DATA_BLOCK "ShiftmodelInterfaceHmi"   // DB103
TITLE = Schichtzeiten / ShiftmodelTimes
AUTHOR : SICAR
FAMILY : Shiftmodel
VERSION : 1.0
// Global DB fuer Schnittstelle HMI / Global DB for HMI interface
// stored: InstanceOfName LSicar_typeShiftmodelHmi, InstanceOfType UDT
"LSicar_typeShiftmodelHmi"
   // VAR RETAIN
   //    shiftTimesListIndex : DInt := 1;
   //    actualTimesDay : Array[0..7] of "LSicar_typeShiftmodTime1Day";
   //    actualSignalsDay : Array[0..7] of "LSicar_typeShiftmodSign1Day";
   //    summary : "LSicar_typeShiftmodSumHmi";
   //    actualDay : USInt := 0;
   //    shiftTimesListOnOff : Bool := TRUE;   // Schichtzeiten Remote OnOff / Shift times OnOff
   //    setAdjTimes : Bool := FALSE;
   //    hmiTimesValidFor : Array[0..3] of "LSicar_typeWeekdayBools";
   //    hmiTimes : Array[0..3] of "LSicar_typeShiftmodTime1Shift";   // Schnittstelle Lokale Zeiten (eingeben am HMI) / Interface Local Times (Input on HMI)
   //    productionTimes : "LSicar_typeProdTimesHmi";
   // END_VAR
BEGIN
   actualTimesDay[0].shift[0..3].endCircuitTime := TOD#00:00:00;
   actualTimesDay[1].shift[0..3].endCircuitTime := TOD#00:00:00;
   actualTimesDay[2].shift[0..3].endCircuitTime := TOD#00:00:00;
   actualTimesDay[3].shift[0..3].endCircuitTime := TOD#00:00:00;
   actualTimesDay[4].shift[0..3].endCircuitTime := TOD#00:00:00;
   actualTimesDay[5].shift[0..3].endCircuitTime := TOD#00:00:00;
   actualTimesDay[6].shift[0..3].endCircuitTime := TOD#00:00:00;
   actualTimesDay[7].shift[0..3].endCircuitTime := TOD#00:00:00;
   actualTimesDay[0].shift[0..3].start := TOD#00:00:00;
   actualTimesDay[1].shift[0..3].start := TOD#00:00:00;
   actualTimesDay[2].shift[0..3].start := TOD#00:00:00;
   actualTimesDay[3].shift[0..3].start := TOD#00:00:00;
   actualTimesDay[4].shift[0..3].start := TOD#00:00:00;
   actualTimesDay[5].shift[0..3].start := TOD#00:00:00;
   actualTimesDay[6].shift[0..3].start := TOD#00:00:00;
   actualTimesDay[7].shift[0..3].start := TOD#00:00:00;
   actualTimesDay[0].shift[0].break[0..4].start := TOD#00:00:00;
   actualTimesDay[0].shift[1].break[0..4].start := TOD#00:00:00;
   actualTimesDay[0].shift[2].break[0..4].start := TOD#00:00:00;
   actualTimesDay[0].shift[3].break[0..4].start := TOD#00:00:00;
   actualTimesDay[1].shift[0].break[0..4].start := TOD#00:00:00;
   actualTimesDay[1].shift[1].break[0..4].start := TOD#00:00:00;
   actualTimesDay[1].shift[2].break[0..4].start := TOD#00:00:00;
   actualTimesDay[1].shift[3].break[0..4].start := TOD#00:00:00;
   actualTimesDay[2].shift[0].break[0..4].start := TOD#00:00:00;
   actualTimesDay[2].shift[1].break[0..4].start := TOD#00:00:00;
   actualTimesDay[2].shift[2].break[0..4].start := TOD#00:00:00;
   actualTimesDay[2].shift[3].break[0..4].start := TOD#00:00:00;
   actualTimesDay[3].shift[0].break[0..4].start := TOD#00:00:00;
   actualTimesDay[3].shift[1].break[0..4].start := TOD#00:00:00;
   actualTimesDay[3].shift[2].break[0..4].start := TOD#00:00:00;
   actualTimesDay[3].shift[3].break[0..4].start := TOD#00:00:00;
   actualTimesDay[4].shift[0].break[0..4].start := TOD#00:00:00;
   actualTimesDay[4].shift[1].break[0..4].start := TOD#00:00:00;
   actualTimesDay[4].shift[2].break[0..4].start := TOD#00:00:00;
   actualTimesDay[4].shift[3].break[0..4].start := TOD#00:00:00;
   actualTimesDay[5].shift[0].break[0..4].start := TOD#00:00:00;
   actualTimesDay[5].shift[1].break[0..4].start := TOD#00:00:00;
   actualTimesDay[5].shift[2].break[0..4].start := TOD#00:00:00;
   actualTimesDay[5].shift[3].break[0..4].start := TOD#00:00:00;
   actualTimesDay[6].shift[0].break[0..4].start := TOD#00:00:00;
   actualTimesDay[6].shift[1].break[0..4].start := TOD#00:00:00;
   actualTimesDay[6].shift[2].break[0..4].start := TOD#00:00:00;
   actualTimesDay[6].shift[3].break[0..4].start := TOD#00:00:00;
   actualTimesDay[7].shift[0].break[0..4].start := TOD#00:00:00;
   actualTimesDay[7].shift[1].break[0..4].start := TOD#00:00:00;
   actualTimesDay[7].shift[2].break[0..4].start := TOD#00:00:00;
   actualTimesDay[7].shift[3].break[0..4].start := TOD#00:00:00;
   actualTimesDay[0].shift[0].break[0..4].startCircuitTime := TOD#00:00:00;
   actualTimesDay[0].shift[1].break[0..4].startCircuitTime := TOD#00:00:00;
   actualTimesDay[0].shift[2].break[0..4].startCircuitTime := TOD#00:00:00;
   actualTimesDay[0].shift[3].break[0..4].startCircuitTime := TOD#00:00:00;
   actualTimesDay[1].shift[0].break[0..4].startCircuitTime := TOD#00:00:00;
   actualTimesDay[1].shift[1].break[0..4].startCircuitTime := TOD#00:00:00;
   actualTimesDay[1].shift[2].break[0..4].startCircuitTime := TOD#00:00:00;
   actualTimesDay[1].shift[3].break[0..4].startCircuitTime := TOD#00:00:00;
   actualTimesDay[2].shift[0].break[0..4].startCircuitTime := TOD#00:00:00;
   actualTimesDay[2].shift[1].break[0..4].startCircuitTime := TOD#00:00:00;
   actualTimesDay[2].shift[2].break[0..4].startCircuitTime := TOD#00:00:00;
   actualTimesDay[2].shift[3].break[0..4].startCircuitTime := TOD#00:00:00;
   actualTimesDay[3].shift[0].break[0..4].startCircuitTime := TOD#00:00:00;
   actualTimesDay[3].shift[1].break[0..4].startCircuitTime := TOD#00:00:00;
   actualTimesDay[3].shift[2].break[0..4].startCircuitTime := TOD#00:00:00;
   actualTimesDay[3].shift[3].break[0..4].startCircuitTime := TOD#00:00:00;
   actualTimesDay[4].shift[0].break[0..4].startCircuitTime := TOD#00:00:00;
   actualTimesDay[4].shift[1].break[0..4].startCircuitTime := TOD#00:00:00;
   actualTimesDay[4].shift[2].break[0..4].startCircuitTime := TOD#00:00:00;
   actualTimesDay[4].shift[3].break[0..4].startCircuitTime := TOD#00:00:00;
   actualTimesDay[5].shift[0].break[0..4].startCircuitTime := TOD#00:00:00;
   actualTimesDay[5].shift[1].break[0..4].startCircuitTime := TOD#00:00:00;
   actualTimesDay[5].shift[2].break[0..4].startCircuitTime := TOD#00:00:00;
   actualTimesDay[5].shift[3].break[0..4].startCircuitTime := TOD#00:00:00;
   actualTimesDay[6].shift[0].break[0..4].startCircuitTime := TOD#00:00:00;
   actualTimesDay[6].shift[1].break[0..4].startCircuitTime := TOD#00:00:00;
   actualTimesDay[6].shift[2].break[0..4].startCircuitTime := TOD#00:00:00;
   actualTimesDay[6].shift[3].break[0..4].startCircuitTime := TOD#00:00:00;
   actualTimesDay[7].shift[0].break[0..4].startCircuitTime := TOD#00:00:00;
   actualTimesDay[7].shift[1].break[0..4].startCircuitTime := TOD#00:00:00;
   actualTimesDay[7].shift[2].break[0..4].startCircuitTime := TOD#00:00:00;
   actualTimesDay[7].shift[3].break[0..4].startCircuitTime := TOD#00:00:00;
   actualTimesDay[0].shift[0].break[0..4].endCircuitTime := TOD#00:00:00;
   actualTimesDay[0].shift[1].break[0..4].endCircuitTime := TOD#00:00:00;
   actualTimesDay[0].shift[2].break[0..4].endCircuitTime := TOD#00:00:00;
   actualTimesDay[0].shift[3].break[0..4].endCircuitTime := TOD#00:00:00;
   actualTimesDay[1].shift[0].break[0..4].endCircuitTime := TOD#00:00:00;
   actualTimesDay[1].shift[1].break[0..4].endCircuitTime := TOD#00:00:00;
   actualTimesDay[1].shift[2].break[0..4].endCircuitTime := TOD#00:00:00;
   actualTimesDay[1].shift[3].break[0..4].endCircuitTime := TOD#00:00:00;
   actualTimesDay[2].shift[0].break[0..4].endCircuitTime := TOD#00:00:00;
   actualTimesDay[2].shift[1].break[0..4].endCircuitTime := TOD#00:00:00;
   actualTimesDay[2].shift[2].break[0..4].endCircuitTime := TOD#00:00:00;
   actualTimesDay[2].shift[3].break[0..4].endCircuitTime := TOD#00:00:00;
   actualTimesDay[3].shift[0].break[0..4].endCircuitTime := TOD#00:00:00;
   actualTimesDay[3].shift[1].break[0..4].endCircuitTime := TOD#00:00:00;
   actualTimesDay[3].shift[2].break[0..4].endCircuitTime := TOD#00:00:00;
   actualTimesDay[3].shift[3].break[0..4].endCircuitTime := TOD#00:00:00;
   actualTimesDay[4].shift[0].break[0..4].endCircuitTime := TOD#00:00:00;
   actualTimesDay[4].shift[1].break[0..4].endCircuitTime := TOD#00:00:00;
   actualTimesDay[4].shift[2].break[0..4].endCircuitTime := TOD#00:00:00;
   actualTimesDay[4].shift[3].break[0..4].endCircuitTime := TOD#00:00:00;
   actualTimesDay[5].shift[0].break[0..4].endCircuitTime := TOD#00:00:00;
   actualTimesDay[5].shift[1].break[0..4].endCircuitTime := TOD#00:00:00;
   actualTimesDay[5].shift[2].break[0..4].endCircuitTime := TOD#00:00:00;
   actualTimesDay[5].shift[3].break[0..4].endCircuitTime := TOD#00:00:00;
   actualTimesDay[6].shift[0].break[0..4].endCircuitTime := TOD#00:00:00;
   actualTimesDay[6].shift[1].break[0..4].endCircuitTime := TOD#00:00:00;
   actualTimesDay[6].shift[2].break[0..4].endCircuitTime := TOD#00:00:00;
   actualTimesDay[6].shift[3].break[0..4].endCircuitTime := TOD#00:00:00;
   actualTimesDay[7].shift[0].break[0..4].endCircuitTime := TOD#00:00:00;
   actualTimesDay[7].shift[1].break[0..4].endCircuitTime := TOD#00:00:00;
   actualTimesDay[7].shift[2].break[0..4].endCircuitTime := TOD#00:00:00;
   actualTimesDay[7].shift[3].break[0..4].endCircuitTime := TOD#00:00:00;
   actualTimesDay[0].shift[0].break[0..4].end := TOD#00:00:00;
   actualTimesDay[0].shift[1].break[0..4].end := TOD#00:00:00;
   actualTimesDay[0].shift[2].break[0..4].end := TOD#00:00:00;
   actualTimesDay[0].shift[3].break[0..4].end := TOD#00:00:00;
   actualTimesDay[1].shift[0].break[0..4].end := TOD#00:00:00;
   actualTimesDay[1].shift[1].break[0..4].end := TOD#00:00:00;
   actualTimesDay[1].shift[2].break[0..4].end := TOD#00:00:00;
   actualTimesDay[1].shift[3].break[0..4].end := TOD#00:00:00;
   actualTimesDay[2].shift[0].break[0..4].end := TOD#00:00:00;
   actualTimesDay[2].shift[1].break[0..4].end := TOD#00:00:00;
   actualTimesDay[2].shift[2].break[0..4].end := TOD#00:00:00;
   actualTimesDay[2].shift[3].break[0..4].end := TOD#00:00:00;
   actualTimesDay[3].shift[0].break[0..4].end := TOD#00:00:00;
   actualTimesDay[3].shift[1].break[0..4].end := TOD#00:00:00;
   actualTimesDay[3].shift[2].break[0..4].end := TOD#00:00:00;
   actualTimesDay[3].shift[3].break[0..4].end := TOD#00:00:00;
   actualTimesDay[4].shift[0].break[0..4].end := TOD#00:00:00;
   actualTimesDay[4].shift[1].break[0..4].end := TOD#00:00:00;
   actualTimesDay[4].shift[2].break[0..4].end := TOD#00:00:00;
   actualTimesDay[4].shift[3].break[0..4].end := TOD#00:00:00;
   actualTimesDay[5].shift[0].break[0..4].end := TOD#00:00:00;
   actualTimesDay[5].shift[1].break[0..4].end := TOD#00:00:00;
   actualTimesDay[5].shift[2].break[0..4].end := TOD#00:00:00;
   actualTimesDay[5].shift[3].break[0..4].end := TOD#00:00:00;
   actualTimesDay[6].shift[0].break[0..4].end := TOD#00:00:00;
   actualTimesDay[6].shift[1].break[0..4].end := TOD#00:00:00;
   actualTimesDay[6].shift[2].break[0..4].end := TOD#00:00:00;
   actualTimesDay[6].shift[3].break[0..4].end := TOD#00:00:00;
   actualTimesDay[7].shift[0].break[0..4].end := TOD#00:00:00;
   actualTimesDay[7].shift[1].break[0..4].end := TOD#00:00:00;
   actualTimesDay[7].shift[2].break[0..4].end := TOD#00:00:00;
   actualTimesDay[7].shift[3].break[0..4].end := TOD#00:00:00;
   actualTimesDay[0].shift[0..3].end := TOD#00:00:00;
   actualTimesDay[1].shift[0..3].end := TOD#00:00:00;
   actualTimesDay[2].shift[0..3].end := TOD#00:00:00;
   actualTimesDay[3].shift[0..3].end := TOD#00:00:00;
   actualTimesDay[4].shift[0..3].end := TOD#00:00:00;
   actualTimesDay[5].shift[0..3].end := TOD#00:00:00;
   actualTimesDay[6].shift[0..3].end := TOD#00:00:00;
   actualTimesDay[7].shift[0..3].end := TOD#00:00:00;
   actualTimesDay[0].shift[0..3].startCircuitTime := TOD#00:00:00;
   actualTimesDay[1].shift[0..3].startCircuitTime := TOD#00:00:00;
   actualTimesDay[2].shift[0..3].startCircuitTime := TOD#00:00:00;
   actualTimesDay[3].shift[0..3].startCircuitTime := TOD#00:00:00;
   actualTimesDay[4].shift[0..3].startCircuitTime := TOD#00:00:00;
   actualTimesDay[5].shift[0..3].startCircuitTime := TOD#00:00:00;
   actualTimesDay[6].shift[0..3].startCircuitTime := TOD#00:00:00;
   actualTimesDay[7].shift[0..3].startCircuitTime := TOD#00:00:00;
   actualSignalsDay[0].shift[0..3].shiftConfig := FALSE;
   actualSignalsDay[1].shift[0..3].shiftConfig := FALSE;
   actualSignalsDay[2].shift[0..3].shiftConfig := FALSE;
   actualSignalsDay[3].shift[0..3].shiftConfig := FALSE;
   actualSignalsDay[4].shift[0..3].shiftConfig := FALSE;
   actualSignalsDay[5].shift[0..3].shiftConfig := FALSE;
   actualSignalsDay[6].shift[0..3].shiftConfig := FALSE;
   actualSignalsDay[7].shift[0..3].shiftConfig := FALSE;
   actualSignalsDay[0].shift[0..3].shiftActive := FALSE;
   actualSignalsDay[1].shift[0..3].shiftActive := FALSE;
   actualSignalsDay[2].shift[0..3].shiftActive := FALSE;
   actualSignalsDay[3].shift[0..3].shiftActive := FALSE;
   actualSignalsDay[4].shift[0..3].shiftActive := FALSE;
   actualSignalsDay[5].shift[0..3].shiftActive := FALSE;
   actualSignalsDay[6].shift[0..3].shiftActive := FALSE;
   actualSignalsDay[7].shift[0..3].shiftActive := FALSE;
   actualSignalsDay[0].shift[0..3].shiftEndCirTimeConfig := FALSE;
   actualSignalsDay[1].shift[0..3].shiftEndCirTimeConfig := FALSE;
   actualSignalsDay[2].shift[0..3].shiftEndCirTimeConfig := FALSE;
   actualSignalsDay[3].shift[0..3].shiftEndCirTimeConfig := FALSE;
   actualSignalsDay[4].shift[0..3].shiftEndCirTimeConfig := FALSE;
   actualSignalsDay[5].shift[0..3].shiftEndCirTimeConfig := FALSE;
   actualSignalsDay[6].shift[0..3].shiftEndCirTimeConfig := FALSE;
   actualSignalsDay[7].shift[0..3].shiftEndCirTimeConfig := FALSE;
   actualSignalsDay[0].shift[0..3].shiftStartCirTimeConfig := FALSE;
   actualSignalsDay[1].shift[0..3].shiftStartCirTimeConfig := FALSE;
   actualSignalsDay[2].shift[0..3].shiftStartCirTimeConfig := FALSE;
   actualSignalsDay[3].shift[0..3].shiftStartCirTimeConfig := FALSE;
   actualSignalsDay[4].shift[0..3].shiftStartCirTimeConfig := FALSE;
   actualSignalsDay[5].shift[0..3].shiftStartCirTimeConfig := FALSE;
   actualSignalsDay[6].shift[0..3].shiftStartCirTimeConfig := FALSE;
   actualSignalsDay[7].shift[0..3].shiftStartCirTimeConfig := FALSE;
   actualSignalsDay[0].shift[0..3].shiftEndCirTimeActive := FALSE;
   actualSignalsDay[1].shift[0..3].shiftEndCirTimeActive := FALSE;
   actualSignalsDay[2].shift[0..3].shiftEndCirTimeActive := FALSE;
   actualSignalsDay[3].shift[0..3].shiftEndCirTimeActive := FALSE;
   actualSignalsDay[4].shift[0..3].shiftEndCirTimeActive := FALSE;
   actualSignalsDay[5].shift[0..3].shiftEndCirTimeActive := FALSE;
   actualSignalsDay[6].shift[0..3].shiftEndCirTimeActive := FALSE;
   actualSignalsDay[7].shift[0..3].shiftEndCirTimeActive := FALSE;
   actualSignalsDay[0].shift[0..3].shiftStartCirTimeActive := FALSE;
   actualSignalsDay[1].shift[0..3].shiftStartCirTimeActive := FALSE;
   actualSignalsDay[2].shift[0..3].shiftStartCirTimeActive := FALSE;
   actualSignalsDay[3].shift[0..3].shiftStartCirTimeActive := FALSE;
   actualSignalsDay[4].shift[0..3].shiftStartCirTimeActive := FALSE;
   actualSignalsDay[5].shift[0..3].shiftStartCirTimeActive := FALSE;
   actualSignalsDay[6].shift[0..3].shiftStartCirTimeActive := FALSE;
   actualSignalsDay[7].shift[0..3].shiftStartCirTimeActive := FALSE;
   actualSignalsDay[0].shift[0..3].shiftSignalsHmi := 16#00;
   actualSignalsDay[1].shift[0..3].shiftSignalsHmi := 16#00;
   actualSignalsDay[2].shift[0..3].shiftSignalsHmi := 16#00;
   actualSignalsDay[3].shift[0..3].shiftSignalsHmi := 16#00;
   actualSignalsDay[4].shift[0..3].shiftSignalsHmi := 16#00;
   actualSignalsDay[5].shift[0..3].shiftSignalsHmi := 16#00;
   actualSignalsDay[6].shift[0..3].shiftSignalsHmi := 16#00;
   actualSignalsDay[7].shift[0..3].shiftSignalsHmi := 16#00;
   actualSignalsDay[0].shift[0].break[0..4].config := FALSE;
   actualSignalsDay[0].shift[1].break[0..4].config := FALSE;
   actualSignalsDay[0].shift[2].break[0..4].config := FALSE;
   actualSignalsDay[0].shift[3].break[0..4].config := FALSE;
   actualSignalsDay[1].shift[0].break[0..4].config := FALSE;
   actualSignalsDay[1].shift[1].break[0..4].config := FALSE;
   actualSignalsDay[1].shift[2].break[0..4].config := FALSE;
   actualSignalsDay[1].shift[3].break[0..4].config := FALSE;
   actualSignalsDay[2].shift[0].break[0..4].config := FALSE;
   actualSignalsDay[2].shift[1].break[0..4].config := FALSE;
   actualSignalsDay[2].shift[2].break[0..4].config := FALSE;
   actualSignalsDay[2].shift[3].break[0..4].config := FALSE;
   actualSignalsDay[3].shift[0].break[0..4].config := FALSE;
   actualSignalsDay[3].shift[1].break[0..4].config := FALSE;
   actualSignalsDay[3].shift[2].break[0..4].config := FALSE;
   actualSignalsDay[3].shift[3].break[0..4].config := FALSE;
   actualSignalsDay[4].shift[0].break[0..4].config := FALSE;
   actualSignalsDay[4].shift[1].break[0..4].config := FALSE;
   actualSignalsDay[4].shift[2].break[0..4].config := FALSE;
   actualSignalsDay[4].shift[3].break[0..4].config := FALSE;
   actualSignalsDay[5].shift[0].break[0..4].config := FALSE;
   actualSignalsDay[5].shift[1].break[0..4].config := FALSE;
   actualSignalsDay[5].shift[2].break[0..4].config := FALSE;
   actualSignalsDay[5].shift[3].break[0..4].config := FALSE;
   actualSignalsDay[6].shift[0].break[0..4].config := FALSE;
   actualSignalsDay[6].shift[1].break[0..4].config := FALSE;
   actualSignalsDay[6].shift[2].break[0..4].config := FALSE;
   actualSignalsDay[6].shift[3].break[0..4].config := FALSE;
   actualSignalsDay[7].shift[0].break[0..4].config := FALSE;
   actualSignalsDay[7].shift[1].break[0..4].config := FALSE;
   actualSignalsDay[7].shift[2].break[0..4].config := FALSE;
   actualSignalsDay[7].shift[3].break[0..4].config := FALSE;
   actualSignalsDay[0].shift[0].break[0..4].active := FALSE;
   actualSignalsDay[0].shift[1].break[0..4].active := FALSE;
   actualSignalsDay[0].shift[2].break[0..4].active := FALSE;
   actualSignalsDay[0].shift[3].break[0..4].active := FALSE;
   actualSignalsDay[1].shift[0].break[0..4].active := FALSE;
   actualSignalsDay[1].shift[1].break[0..4].active := FALSE;
   actualSignalsDay[1].shift[2].break[0..4].active := FALSE;
   actualSignalsDay[1].shift[3].break[0..4].active := FALSE;
   actualSignalsDay[2].shift[0].break[0..4].active := FALSE;
   actualSignalsDay[2].shift[1].break[0..4].active := FALSE;
   actualSignalsDay[2].shift[2].break[0..4].active := FALSE;
   actualSignalsDay[2].shift[3].break[0..4].active := FALSE;
   actualSignalsDay[3].shift[0].break[0..4].active := FALSE;
   actualSignalsDay[3].shift[1].break[0..4].active := FALSE;
   actualSignalsDay[3].shift[2].break[0..4].active := FALSE;
   actualSignalsDay[3].shift[3].break[0..4].active := FALSE;
   actualSignalsDay[4].shift[0].break[0..4].active := FALSE;
   actualSignalsDay[4].shift[1].break[0..4].active := FALSE;
   actualSignalsDay[4].shift[2].break[0..4].active := FALSE;
   actualSignalsDay[4].shift[3].break[0..4].active := FALSE;
   actualSignalsDay[5].shift[0].break[0..4].active := FALSE;
   actualSignalsDay[5].shift[1].break[0..4].active := FALSE;
   actualSignalsDay[5].shift[2].break[0..4].active := FALSE;
   actualSignalsDay[5].shift[3].break[0..4].active := FALSE;
   actualSignalsDay[6].shift[0].break[0..4].active := FALSE;
   actualSignalsDay[6].shift[1].break[0..4].active := FALSE;
   actualSignalsDay[6].shift[2].break[0..4].active := FALSE;
   actualSignalsDay[6].shift[3].break[0..4].active := FALSE;
   actualSignalsDay[7].shift[0].break[0..4].active := FALSE;
   actualSignalsDay[7].shift[1].break[0..4].active := FALSE;
   actualSignalsDay[7].shift[2].break[0..4].active := FALSE;
   actualSignalsDay[7].shift[3].break[0..4].active := FALSE;
   actualSignalsDay[0].shift[0].break[0..4].circuitTimeConfig := FALSE;
   actualSignalsDay[0].shift[1].break[0..4].circuitTimeConfig := FALSE;
   actualSignalsDay[0].shift[2].break[0..4].circuitTimeConfig := FALSE;
   actualSignalsDay[0].shift[3].break[0..4].circuitTimeConfig := FALSE;
   actualSignalsDay[1].shift[0].break[0..4].circuitTimeConfig := FALSE;
   actualSignalsDay[1].shift[1].break[0..4].circuitTimeConfig := FALSE;
   actualSignalsDay[1].shift[2].break[0..4].circuitTimeConfig := FALSE;
   actualSignalsDay[1].shift[3].break[0..4].circuitTimeConfig := FALSE;
   actualSignalsDay[2].shift[0].break[0..4].circuitTimeConfig := FALSE;
   actualSignalsDay[2].shift[1].break[0..4].circuitTimeConfig := FALSE;
   actualSignalsDay[2].shift[2].break[0..4].circuitTimeConfig := FALSE;
   actualSignalsDay[2].shift[3].break[0..4].circuitTimeConfig := FALSE;
   actualSignalsDay[3].shift[0].break[0..4].circuitTimeConfig := FALSE;
   actualSignalsDay[3].shift[1].break[0..4].circuitTimeConfig := FALSE;
   actualSignalsDay[3].shift[2].break[0..4].circuitTimeConfig := FALSE;
   actualSignalsDay[3].shift[3].break[0..4].circuitTimeConfig := FALSE;
   actualSignalsDay[4].shift[0].break[0..4].circuitTimeConfig := FALSE;
   actualSignalsDay[4].shift[1].break[0..4].circuitTimeConfig := FALSE;
   actualSignalsDay[4].shift[2].break[0..4].circuitTimeConfig := FALSE;
   actualSignalsDay[4].shift[3].break[0..4].circuitTimeConfig := FALSE;
   actualSignalsDay[5].shift[0].break[0..4].circuitTimeConfig := FALSE;
   actualSignalsDay[5].shift[1].break[0..4].circuitTimeConfig := FALSE;
   actualSignalsDay[5].shift[2].break[0..4].circuitTimeConfig := FALSE;
   actualSignalsDay[5].shift[3].break[0..4].circuitTimeConfig := FALSE;
   actualSignalsDay[6].shift[0].break[0..4].circuitTimeConfig := FALSE;
   actualSignalsDay[6].shift[1].break[0..4].circuitTimeConfig := FALSE;
   actualSignalsDay[6].shift[2].break[0..4].circuitTimeConfig := FALSE;
   actualSignalsDay[6].shift[3].break[0..4].circuitTimeConfig := FALSE;
   actualSignalsDay[7].shift[0].break[0..4].circuitTimeConfig := FALSE;
   actualSignalsDay[7].shift[1].break[0..4].circuitTimeConfig := FALSE;
   actualSignalsDay[7].shift[2].break[0..4].circuitTimeConfig := FALSE;
   actualSignalsDay[7].shift[3].break[0..4].circuitTimeConfig := FALSE;
   actualSignalsDay[0].shift[0].break[0..4].circuitTimeActive := FALSE;
   actualSignalsDay[0].shift[1].break[0..4].circuitTimeActive := FALSE;
   actualSignalsDay[0].shift[2].break[0..4].circuitTimeActive := FALSE;
   actualSignalsDay[0].shift[3].break[0..4].circuitTimeActive := FALSE;
   actualSignalsDay[1].shift[0].break[0..4].circuitTimeActive := FALSE;
   actualSignalsDay[1].shift[1].break[0..4].circuitTimeActive := FALSE;
   actualSignalsDay[1].shift[2].break[0..4].circuitTimeActive := FALSE;
   actualSignalsDay[1].shift[3].break[0..4].circuitTimeActive := FALSE;
   actualSignalsDay[2].shift[0].break[0..4].circuitTimeActive := FALSE;
   actualSignalsDay[2].shift[1].break[0..4].circuitTimeActive := FALSE;
   actualSignalsDay[2].shift[2].break[0..4].circuitTimeActive := FALSE;
   actualSignalsDay[2].shift[3].break[0..4].circuitTimeActive := FALSE;
   actualSignalsDay[3].shift[0].break[0..4].circuitTimeActive := FALSE;
   actualSignalsDay[3].shift[1].break[0..4].circuitTimeActive := FALSE;
   actualSignalsDay[3].shift[2].break[0..4].circuitTimeActive := FALSE;
   actualSignalsDay[3].shift[3].break[0..4].circuitTimeActive := FALSE;
   actualSignalsDay[4].shift[0].break[0..4].circuitTimeActive := FALSE;
   actualSignalsDay[4].shift[1].break[0..4].circuitTimeActive := FALSE;
   actualSignalsDay[4].shift[2].break[0..4].circuitTimeActive := FALSE;
   actualSignalsDay[4].shift[3].break[0..4].circuitTimeActive := FALSE;
   actualSignalsDay[5].shift[0].break[0..4].circuitTimeActive := FALSE;
   actualSignalsDay[5].shift[1].break[0..4].circuitTimeActive := FALSE;
   actualSignalsDay[5].shift[2].break[0..4].circuitTimeActive := FALSE;
   actualSignalsDay[5].shift[3].break[0..4].circuitTimeActive := FALSE;
   actualSignalsDay[6].shift[0].break[0..4].circuitTimeActive := FALSE;
   actualSignalsDay[6].shift[1].break[0..4].circuitTimeActive := FALSE;
   actualSignalsDay[6].shift[2].break[0..4].circuitTimeActive := FALSE;
   actualSignalsDay[6].shift[3].break[0..4].circuitTimeActive := FALSE;
   actualSignalsDay[7].shift[0].break[0..4].circuitTimeActive := FALSE;
   actualSignalsDay[7].shift[1].break[0..4].circuitTimeActive := FALSE;
   actualSignalsDay[7].shift[2].break[0..4].circuitTimeActive := FALSE;
   actualSignalsDay[7].shift[3].break[0..4].circuitTimeActive := FALSE;
   actualSignalsDay[0].shift[0..3].breakSignalsHmi := 16#0000;
   actualSignalsDay[1].shift[0..3].breakSignalsHmi := 16#0000;
   actualSignalsDay[2].shift[0..3].breakSignalsHmi := 16#0000;
   actualSignalsDay[3].shift[0..3].breakSignalsHmi := 16#0000;
   actualSignalsDay[4].shift[0..3].breakSignalsHmi := 16#0000;
   actualSignalsDay[5].shift[0..3].breakSignalsHmi := 16#0000;
   actualSignalsDay[6].shift[0..3].breakSignalsHmi := 16#0000;
   actualSignalsDay[7].shift[0..3].breakSignalsHmi := 16#0000;
   actualSignalsDay[0..7].shiftsPerDay := 0;
   summary.earlyShiftActive := FALSE;
   summary.lateShiftActive := FALSE;
   summary.nightShiftActive := FALSE;
   summary.breakInShiftActive := FALSE;
   summary.breakBetweenShiftAct := FALSE;
   summary.breakActive := FALSE;
   summary.circuitTimeInShiftAct := FALSE;
   summary.circuitTimeBetwShiftAct := FALSE;
   summary.circuitTimeActive := FALSE;
   summary.noOfWorkdays := 0;
   summary.workdays[0..7] := FALSE;
   hmiTimesValidFor[0..3].sunday := FALSE;
   hmiTimesValidFor[0..3].monday := FALSE;
   hmiTimesValidFor[0..3].tuesday := FALSE;
   hmiTimesValidFor[0..3].wednesday := FALSE;
   hmiTimesValidFor[0..3].thursday := FALSE;
   hmiTimesValidFor[0..3].friday := FALSE;
   hmiTimesValidFor[0..3].saturday := FALSE;
   hmiTimes[0].endCircuitTime := TOD#00:00:00;
   hmiTimes[1].endCircuitTime := TOD#05:57:00;
   hmiTimes[2].endCircuitTime := TOD#13:57:00;
   hmiTimes[3].endCircuitTime := TOD#21:57:00;
   hmiTimes[0].start := TOD#00:00:00;
   hmiTimes[1].start := TOD#06:00:00;
   hmiTimes[2].start := TOD#14:00:00;
   hmiTimes[3].start := TOD#22:00:00;
   hmiTimes[0].break[0..4].start := TOD#00:00:00;
   hmiTimes[1].break[0].start := TOD#00:00:00;
   hmiTimes[1].break[1].start := TOD#08:00:00;
   hmiTimes[1].break[2].start := TOD#10:00:00;
   hmiTimes[1].break[3].start := TOD#12:00:00;
   hmiTimes[1].break[4].start := TOD#00:00:00;
   hmiTimes[2].break[0].start := TOD#00:00:00;
   hmiTimes[2].break[1].start := TOD#16:00:00;
   hmiTimes[2].break[2].start := TOD#18:00:00;
   hmiTimes[2].break[3].start := TOD#20:00:00;
   hmiTimes[2].break[4].start := TOD#00:00:00;
   hmiTimes[3].break[0..1].start := TOD#00:00:00;
   hmiTimes[3].break[2].start := TOD#02:00:00;
   hmiTimes[3].break[3].start := TOD#04:00:00;
   hmiTimes[3].break[4].start := TOD#00:00:00;
   hmiTimes[0].break[0..4].startCircuitTime := TOD#00:00:00;
   hmiTimes[1].break[0].startCircuitTime := TOD#00:00:00;
   hmiTimes[1].break[1].startCircuitTime := TOD#08:02:00;
   hmiTimes[1].break[2].startCircuitTime := TOD#00:00:00;
   hmiTimes[1].break[3].startCircuitTime := TOD#12:02:00;
   hmiTimes[1].break[4].startCircuitTime := TOD#00:00:00;
   hmiTimes[2].break[0].startCircuitTime := TOD#00:00:00;
   hmiTimes[2].break[1].startCircuitTime := TOD#16:02:00;
   hmiTimes[2].break[2].startCircuitTime := TOD#00:00:00;
   hmiTimes[2].break[3].startCircuitTime := TOD#20:02:00;
   hmiTimes[2].break[4].startCircuitTime := TOD#00:00:00;
   hmiTimes[3].break[0].startCircuitTime := TOD#00:00:00;
   hmiTimes[3].break[1].startCircuitTime := TOD#00:02:00;
   hmiTimes[3].break[2].startCircuitTime := TOD#00:00:00;
   hmiTimes[3].break[3].startCircuitTime := TOD#04:02:00;
   hmiTimes[3].break[4].startCircuitTime := TOD#00:00:00;
   hmiTimes[0].break[0..4].endCircuitTime := TOD#00:00:00;
   hmiTimes[1].break[0].endCircuitTime := TOD#00:00:00;
   hmiTimes[1].break[1].endCircuitTime := TOD#08:13:00;
   hmiTimes[1].break[2].endCircuitTime := TOD#00:00:00;
   hmiTimes[1].break[3].endCircuitTime := TOD#12:13:00;
   hmiTimes[1].break[4].endCircuitTime := TOD#00:00:00;
   hmiTimes[2].break[0].endCircuitTime := TOD#00:00:00;
   hmiTimes[2].break[1].endCircuitTime := TOD#16:13:00;
   hmiTimes[2].break[2].endCircuitTime := TOD#00:00:00;
   hmiTimes[2].break[3].endCircuitTime := TOD#20:13:00;
   hmiTimes[2].break[4].endCircuitTime := TOD#00:00:00;
   hmiTimes[3].break[0].endCircuitTime := TOD#00:00:00;
   hmiTimes[3].break[1].endCircuitTime := TOD#00:13:00;
   hmiTimes[3].break[2].endCircuitTime := TOD#00:00:00;
   hmiTimes[3].break[3].endCircuitTime := TOD#04:13:00;
   hmiTimes[3].break[4].endCircuitTime := TOD#00:00:00;
   hmiTimes[0].break[0..4].end := TOD#00:00:00;
   hmiTimes[1].break[0].end := TOD#00:00:00;
   hmiTimes[1].break[1].end := TOD#08:15:00;
   hmiTimes[1].break[2].end := TOD#10:10:00;
   hmiTimes[1].break[3].end := TOD#12:15:00;
   hmiTimes[1].break[4].end := TOD#00:00:00;
   hmiTimes[2].break[0].end := TOD#00:00:00;
   hmiTimes[2].break[1].end := TOD#16:15:00;
   hmiTimes[2].break[2].end := TOD#18:10:00;
   hmiTimes[2].break[3].end := TOD#20:15:00;
   hmiTimes[2].break[4].end := TOD#00:00:00;
   hmiTimes[3].break[0].end := TOD#00:00:00;
   hmiTimes[3].break[1].end := TOD#00:15:00;
   hmiTimes[3].break[2].end := TOD#02:10:00;
   hmiTimes[3].break[3].end := TOD#04:15:00;
   hmiTimes[3].break[4].end := TOD#00:00:00;
   hmiTimes[0].end := TOD#00:00:00;
   hmiTimes[1].end := TOD#13:30:00;
   hmiTimes[2].end := TOD#21:30:00;
   hmiTimes[3].end := TOD#05:30:00;
   hmiTimes[0].startCircuitTime := TOD#00:00:00;
   hmiTimes[1].startCircuitTime := TOD#13:33:00;
   hmiTimes[2].startCircuitTime := TOD#21:33:00;
   hmiTimes[3].startCircuitTime := TOD#05:33:00;
   productionTimes.currentShiftTimes.start := TOD#00:00:00;
   productionTimes.currentShiftTimes.break[0..4].start := TOD#00:00:00;
   productionTimes.currentShiftTimes.break[0..4].startCircuitTime := TOD#00:00:00;
   productionTimes.currentShiftTimes.break[0..4].endCircuitTime := TOD#00:00:00;
   productionTimes.currentShiftTimes.break[0..4].end := TOD#00:00:00;
   productionTimes.currentShiftTimes.end := TOD#00:00:00;
   productionTimes.prodTimeTarget := TOD#00:00:00;
   productionTimes.prodTimeTargetTime := T#0MS;
   productionTimes.prodTimeExpired := TOD#00:00:00;
   productionTimes.prodTimeExpiredTime := T#0MS;
   productionTimes.breakActSum := FALSE;
   productionTimes.shiftActive := FALSE;
END_DATA_BLOCK

DATA_BLOCK "CallSimulation_DB"   // DB57
// stored: InstanceOfName CallSimulation, InstanceOfType FB
"CallSimulation"
BEGIN
END_DATA_BLOCK

DATA_BLOCK "InstCallGlobal"   // DB265
// stored: InstanceOfName CallGlobal, InstanceOfType FB
"CallGlobal"
BEGIN
   instLAF_PowerOnOff.on := FALSE;
   instLAF_PowerOnOff.off := FALSE;
   instLAF_PowerOnOff.powerStatus := 0;
   instLAF_PowerOnOff.enablePower := FALSE;
   instLAF_PowerOnOff.statMemOn := FALSE;
   instLAF_HmiHeaderManager.statFirstCall := FALSE;
   instLAF_HmiHeaderManager.statLowerBoundUnit := 0;
   instLAF_HmiHeaderManager.statUpperBoundUnit := 0;
   instLAF_HmiHeaderManager.statLowerBoundHmi := 0;
   instLAF_HmiHeaderManager.statUpperBoundHmi := 1;
   instLAF_ClockGen.clk10Hz := TRUE;
   instLAF_ClockGen.clk5Hz := TRUE;
   instLAF_ClockGen.clk2Hz5 := FALSE;
   instLAF_ClockGen.clk2Hz := TRUE;
   instLAF_ClockGen.clk1Hz25 := FALSE;
   instLAF_ClockGen.clk1Hz := TRUE;
   instLAF_ClockGen.clk0Hz625 := TRUE;
   instLAF_ClockGen.clk0Hz5 := FALSE;
   instLAF_ClockGen.statMemRuntime := 2.78088143015202E-308;
   instLAF_ClockGen.statCalcTimeClk10Hz := 18157;
   instLAF_ClockGen.statCalcTimeClk5Hz := 18157;
   instLAF_ClockGen.statCalcTimeClk2Hz5 := 18157;
   instLAF_ClockGen.statCalcTimeClk2Hz := 18157;
   instLAF_ClockGen.statCalcTimeClk1Hz25 := 218157;
   instLAF_ClockGen.statCalcTimeClk1Hz := 18157;
   instLAF_ClockGen.statCalcTimeClk0Hz625 := 618157;
   instLAF_ClockGen.statCalcTimeClk0Hz5 := 18157;
   instLAF_ClockGen.statStateFlagClk10Hz := FALSE;
   instLAF_ClockGen.statStateFlagClk5Hz := FALSE;
   instLAF_ClockGen.statStateFlagClk2Hz5 := TRUE;
   instLAF_ClockGen.statStateFlagClk2Hz := FALSE;
   instLAF_ClockGen.statStateFlagClk1Hz25 := TRUE;
   instLAF_ClockGen.statStateFlagClk1Hz := FALSE;
   instLAF_ClockGen.statStateFlagClk0Hz625 := FALSE;
   instLAF_ClockGen.statStateFlagClk0Hz5 := TRUE;
   instLSNTP_Server.enable := true;
   instLSNTP_Server.connID := 16#0085;
   instLSNTP_Server.referenceID := 0;
   instLSNTP_Server.lastTimeSet := DTL#1990-01-01-00:00:00;
   instLSNTP_Server.valid := TRUE;
   instLSNTP_Server.busy := TRUE;
   instLSNTP_Server.error := FALSE;
   instLSNTP_Server.status := 16#7002;
   instLSNTP_Server.diagnostics.status := 16#0000;
   instLSNTP_Server.diagnostics.subfunctionStatus := 16#0000_0000;
   instLSNTP_Server.diagnostics.stateNumber := 0;
   instLSNTP_Server.statEnableOld := TRUE;
   instLSNTP_Server.statValid := TRUE;
   instLSNTP_Server.statBusy := TRUE;
   instLSNTP_Server.statError := FALSE;
   instLSNTP_Server.statErrorUserCleared := FALSE;
   instLSNTP_Server.statErrorAutoCleared := FALSE;
   instLSNTP_Server.statStatus := 16#7002;
   instLSNTP_Server.statSubfunctionStatus := 16#0000;
   instLSNTP_Server.statFBErrorState := 0;
   instLSNTP_Server.statFBState := 50;
   instLSNTP_Server.statDisablingCompleted := FALSE;
   instLSNTP_Server.statEmptyDiagnostics.status := 16#0000;
   instLSNTP_Server.statEmptyDiagnostics.subfunctionStatus := 16#0000_0000;
   instLSNTP_Server.statEmptyDiagnostics.stateNumber := 0;
   instLSNTP_Server.instTCon.REQ := TRUE;
   instLSNTP_Server.instTCon.ID := 16#0085;
   instLSNTP_Server.instTCon.DONE := TRUE;
   instLSNTP_Server.instTCon.BUSY := FALSE;
   instLSNTP_Server.instTCon.ERROR := FALSE;
   instLSNTP_Server.instTCon.STATUS := 16#0000;
   instLSNTP_Server.instTURcv.ID := 16#0085;
   instLSNTP_Server.instTURcv.LEN := 0;
   instLSNTP_Server.instTURcv.ADHOC := FALSE;
   instLSNTP_Server.instTURcv.NDR := FALSE;
   instLSNTP_Server.instTURcv.BUSY := TRUE;
   instLSNTP_Server.instTURcv.ERROR := FALSE;
   instLSNTP_Server.instTURcv.STATUS := 16#7002;
   instLSNTP_Server.instTURcv.RCVD_LEN := 0;
   instLSNTP_Server.instTUSend.REQ := FALSE;
   instLSNTP_Server.instTUSend.ID := 16#0000;
   instLSNTP_Server.instTUSend.LEN := 0;
   instLSNTP_Server.instTUSend.DONE := FALSE;
   instLSNTP_Server.instTUSend.BUSY := FALSE;
   instLSNTP_Server.instTUSend.ERROR := FALSE;
   instLSNTP_Server.instTUSend.STATUS := 16#7000;
   instLSNTP_Server.instTDiscon.REQ := FALSE;
   instLSNTP_Server.instTDiscon.ID := 16#0000;
   instLSNTP_Server.instTDiscon.DONE := FALSE;
   instLSNTP_Server.instTDiscon.BUSY := FALSE;
   instLSNTP_Server.instTDiscon.ERROR := FALSE;
   instLSNTP_Server.instTDiscon.STATUS := 16#7000;
   instLSNTP_Server.statConParam.InterfaceId := 72;
   instLSNTP_Server.statConParam.ID := 16#0085;
   instLSNTP_Server.statConParam.ConnectionType := 16#13;
   instLSNTP_Server.statConParam.ActiveEstablished := FALSE;
   instLSNTP_Server.statConParam.RemoteAddress.ADDR[1..4] := 16#00;
   instLSNTP_Server.statConParam.RemotePort := 0;
   instLSNTP_Server.statConParam.LocalPort := 123;
   instLSNTP_Server.statAddr.REM_IP_ADDR[1..4] := 0;
   instLSNTP_Server.statAddr.REM_PORT_NR := 0;
   instLSNTP_Server.statAddr.RESERVED := 16#0000;
   instLSNTP_Server.statTelegramRcvd.flags[0..3] := 16#00;
   instLSNTP_Server.statTelegramRcvd.rootDelay := 16#0000_0000;
   instLSNTP_Server.statTelegramRcvd.rootDispersion := 16#0000_0000;
   instLSNTP_Server.statTelegramRcvd.referenceId[0..3] := ' ';
   instLSNTP_Server.statTelegramRcvd.timestamps.reference.sec := 16#0000_0000;
   instLSNTP_Server.statTelegramRcvd.timestamps.reference.secFrac := 16#0000_0000;
   instLSNTP_Server.statTelegramRcvd.timestamps.originate.sec := 16#0000_0000;
   instLSNTP_Server.statTelegramRcvd.timestamps.originate.secFrac := 16#0000_0000;
   instLSNTP_Server.statTelegramRcvd.timestamps.receive.sec := 16#0000_0000;
   instLSNTP_Server.statTelegramRcvd.timestamps.receive.secFrac := 16#0000_0000;
   instLSNTP_Server.statTelegramRcvd.timestamps.transmit.sec := 16#0000_0000;
   instLSNTP_Server.statTelegramRcvd.timestamps.transmit.secFrac := 16#0000_0000;
   instLSNTP_Server.statTelegramRcvd.keyIdentifier := 16#0000_0000;
   instLSNTP_Server.statTelegramRcvd.messageDigest[0..15] := 16#00;
   instLSNTP_Server.statTelegramSend.flags[0..3] := 16#00;
   instLSNTP_Server.statTelegramSend.rootDelay := 16#0000_0000;
   instLSNTP_Server.statTelegramSend.rootDispersion := 16#0000_0000;
   instLSNTP_Server.statTelegramSend.referenceId[0..3] := ' ';
   instLSNTP_Server.statTelegramSend.timestamps.reference.sec := 16#0000_0000;
   instLSNTP_Server.statTelegramSend.timestamps.reference.secFrac := 16#0000_0000;
   instLSNTP_Server.statTelegramSend.timestamps.originate.sec := 16#0000_0000;
   instLSNTP_Server.statTelegramSend.timestamps.originate.secFrac := 16#0000_0000;
   instLSNTP_Server.statTelegramSend.timestamps.receive.sec := 16#0000_0000;
   instLSNTP_Server.statTelegramSend.timestamps.receive.secFrac := 16#0000_0000;
   instLSNTP_Server.statTelegramSend.timestamps.transmit.sec := 16#0000_0000;
   instLSNTP_Server.statTelegramSend.timestamps.transmit.secFrac := 16#0000_0000;
   instLSNTP_Server.statTelegramSend.keyIdentifier := 16#0000_0000;
   instLSNTP_Server.statTelegramSend.messageDigest[0..15] := 16#00;
   instRemoteAccess.lifebitMpPlc := 5;
   instRemoteAccess.connectionTimeOut := T#5S;
   instRemoteAccess.ucpPointerDisabled := FALSE;
   instRemoteAccess.status := 16#0000;
   instRemoteAccess.error := FALSE;
   instRemoteAccess.connectionEnded := FALSE;
   instRemoteAccess.keySwitchMp := 0;
   instRemoteAccess.readoutBoxIdPanel := 0;
   instRemoteAccess.statFirstCall := FALSE;
   instRemoteAccess.statPreviousLifebit := 5;
   instRemoteAccess.statEndConn := FALSE;
   instRemoteAccess.statStatus := 16#0000;
   instRemoteAccess.statLowerBound := 1;
   instRemoteAccess.statUpperBound := 2;
   instRemoteAccess.instTimerLifebit.PT := T#5S;
   instRemoteAccess.instTimerLifebit.IN := TRUE;
END_DATA_BLOCK

DATA_BLOCK "instRecipe"   // DB486
// stored: InstanceOfName LER_Recipe, InstanceOfType FB
"LER_Recipe"
   // VAR_INPUT
   //    enable : Bool;
   //    applyBT : Bool;
   // END_VAR
   // VAR_IN_OUT
   //    parameterRecipeInterface : "HMI_IF_Parameter_LIstRecipe_Interface";
   //    parameterListSV : "HMI_IF_Parameter_ListRecipe_UDT";
   //    parameterListPV : "HMI_IF_Parameter_ListRecipe_UDT";
   // END_VAR
BEGIN
END_DATA_BLOCK

DATA_BLOCK "instTeachingPosAnodeAlignTableAxisX"   // DB453
// stored: InstanceOfName LER_TeachingPos_Interface, InstanceOfType FB
"LER_TeachingPos_Interface"
   // VAR_INPUT
   //    enable : Bool;
   //    selectTeachingPos : SInt;
   //    indexTeachingPos : SInt;
   // END_VAR
   // VAR_IN_OUT
   //    configurationSetPositions : Array[0..15] of "LBC_typeAxis64PosSetPosition";
   //    moduleInterface : "LBC_typeAxis64PosInterface";
   //    hmiInterface : Array[0..48] of "LER_TypeTeachingPosInterface";
   // END_VAR
   // VAR
   //    statPulse : Array[0..9] of Bool;
   //    statTonTimer : Array[0..15] of TON_TIME;
   //    statLastTeachingPosIndex : SInt;
   // END_VAR
BEGIN
END_DATA_BLOCK

DATA_BLOCK "instTeachingPosAnodeAlignTableAxisY1"   // DB461
// stored: InstanceOfName LER_TeachingPos_Interface, InstanceOfType FB
"LER_TeachingPos_Interface"
   // VAR_INPUT
   //    enable : Bool;
   //    selectTeachingPos : SInt;
   //    indexTeachingPos : SInt;
   // END_VAR
   // VAR_IN_OUT
   //    configurationSetPositions : Array[0..15] of "LBC_typeAxis64PosSetPosition";
   //    moduleInterface : "LBC_typeAxis64PosInterface";
   //    hmiInterface : Array[0..48] of "LER_TypeTeachingPosInterface";
   // END_VAR
   // VAR
   //    statPulse : Array[0..9] of Bool;
   //    statTonTimer : Array[0..15] of TON_TIME;
   //    statLastTeachingPosIndex : SInt;
   // END_VAR
BEGIN
END_DATA_BLOCK

DATA_BLOCK "instTeachingPosAnodeAlignTableAxisY2"   // DB460
// stored: InstanceOfName LER_TeachingPos_Interface, InstanceOfType FB
"LER_TeachingPos_Interface"
   // VAR_INPUT
   //    enable : Bool;
   //    selectTeachingPos : SInt;
   //    indexTeachingPos : SInt;
   // END_VAR
   // VAR_IN_OUT
   //    configurationSetPositions : Array[0..15] of "LBC_typeAxis64PosSetPosition";
   //    moduleInterface : "LBC_typeAxis64PosInterface";
   //    hmiInterface : Array[0..48] of "LER_TypeTeachingPosInterface";
   // END_VAR
   // VAR
   //    statPulse : Array[0..9] of Bool;
   //    statTonTimer : Array[0..15] of TON_TIME;
   //    statLastTeachingPosIndex : SInt;
   // END_VAR
BEGIN
END_DATA_BLOCK

DATA_BLOCK "instTeachingPosAnodeMainPnP1AxisX"   // DB271
// stored: InstanceOfName LER_TeachingPos_Interface, InstanceOfType FB
"LER_TeachingPos_Interface"
   // VAR_INPUT
   //    enable : Bool;
   //    selectTeachingPos : SInt;
   //    indexTeachingPos : SInt;
   // END_VAR
   // VAR_IN_OUT
   //    configurationSetPositions : Array[0..15] of "LBC_typeAxis64PosSetPosition";
   //    moduleInterface : "LBC_typeAxis64PosInterface";
   //    hmiInterface : Array[0..48] of "LER_TypeTeachingPosInterface";
   // END_VAR
   // VAR
   //    statPulse : Array[0..9] of Bool;
   //    statTonTimer : Array[0..15] of TON_TIME;
   //    statLastTeachingPosIndex : SInt;
   // END_VAR
BEGIN
END_DATA_BLOCK

DATA_BLOCK "instTeachingPosAnodeMainPnP1AxisY"   // DB355
// stored: InstanceOfName LER_TeachingPos_Interface, InstanceOfType FB
"LER_TeachingPos_Interface"
   // VAR_INPUT
   //    enable : Bool;
   //    selectTeachingPos : SInt;
   //    indexTeachingPos : SInt;
   // END_VAR
   // VAR_IN_OUT
   //    configurationSetPositions : Array[0..15] of "LBC_typeAxis64PosSetPosition";
   //    moduleInterface : "LBC_typeAxis64PosInterface";
   //    hmiInterface : Array[0..48] of "LER_TypeTeachingPosInterface";
   // END_VAR
   // VAR
   //    statPulse : Array[0..9] of Bool;
   //    statTonTimer : Array[0..15] of TON_TIME;
   //    statLastTeachingPosIndex : SInt;
   // END_VAR
BEGIN
END_DATA_BLOCK

DATA_BLOCK "instTeachingPosAnodeMainPnP1AxisZ"   // DB356
// stored: InstanceOfName LER_TeachingPos_Interface, InstanceOfType FB
"LER_TeachingPos_Interface"
   // VAR_INPUT
   //    enable : Bool;
   //    selectTeachingPos : SInt;
   //    indexTeachingPos : SInt;
   // END_VAR
   // VAR_IN_OUT
   //    configurationSetPositions : Array[0..15] of "LBC_typeAxis64PosSetPosition";
   //    moduleInterface : "LBC_typeAxis64PosInterface";
   //    hmiInterface : Array[0..48] of "LER_TypeTeachingPosInterface";
   // END_VAR
   // VAR
   //    statPulse : Array[0..9] of Bool;
   //    statTonTimer : Array[0..15] of TON_TIME;
   //    statLastTeachingPosIndex : SInt;
   // END_VAR
BEGIN
END_DATA_BLOCK

DATA_BLOCK "instTeachingPosAnodeMainPnP2AxisX"   // DB277
// stored: InstanceOfName LER_TeachingPos_Interface, InstanceOfType FB
"LER_TeachingPos_Interface"
   // VAR_INPUT
   //    enable : Bool;
   //    selectTeachingPos : SInt;
   //    indexTeachingPos : SInt;
   // END_VAR
   // VAR_IN_OUT
   //    configurationSetPositions : Array[0..15] of "LBC_typeAxis64PosSetPosition";
   //    moduleInterface : "LBC_typeAxis64PosInterface";
   //    hmiInterface : Array[0..48] of "LER_TypeTeachingPosInterface";
   // END_VAR
   // VAR
   //    statPulse : Array[0..9] of Bool;
   //    statTonTimer : Array[0..15] of TON_TIME;
   //    statLastTeachingPosIndex : SInt;
   // END_VAR
BEGIN
END_DATA_BLOCK

DATA_BLOCK "instTeachingPosAnodeMainPnP2AxisZ"   // DB452
// stored: InstanceOfName LER_TeachingPos_Interface, InstanceOfType FB
"LER_TeachingPos_Interface"
   // VAR_INPUT
   //    enable : Bool;
   //    selectTeachingPos : SInt;
   //    indexTeachingPos : SInt;
   // END_VAR
   // VAR_IN_OUT
   //    configurationSetPositions : Array[0..15] of "LBC_typeAxis64PosSetPosition";
   //    moduleInterface : "LBC_typeAxis64PosInterface";
   //    hmiInterface : Array[0..48] of "LER_TypeTeachingPosInterface";
   // END_VAR
   // VAR
   //    statPulse : Array[0..9] of Bool;
   //    statTonTimer : Array[0..15] of TON_TIME;
   //    statLastTeachingPosIndex : SInt;
   // END_VAR
BEGIN
END_DATA_BLOCK

DATA_BLOCK "instTeachingPosCathodeAlignTableAxisX"   // DB462
// stored: InstanceOfName LER_TeachingPos_Interface, InstanceOfType FB
"LER_TeachingPos_Interface"
   // VAR_INPUT
   //    enable : Bool;
   //    selectTeachingPos : SInt;
   //    indexTeachingPos : SInt;
   // END_VAR
   // VAR_IN_OUT
   //    configurationSetPositions : Array[0..15] of "LBC_typeAxis64PosSetPosition";
   //    moduleInterface : "LBC_typeAxis64PosInterface";
   //    hmiInterface : Array[0..48] of "LER_TypeTeachingPosInterface";
   // END_VAR
   // VAR
   //    statPulse : Array[0..9] of Bool;
   //    statTonTimer : Array[0..15] of TON_TIME;
   //    statLastTeachingPosIndex : SInt;
   // END_VAR
BEGIN
END_DATA_BLOCK

DATA_BLOCK "instTeachingPosCathodeAlignTableAxisY1"   // DB463
// stored: InstanceOfName LER_TeachingPos_Interface, InstanceOfType FB
"LER_TeachingPos_Interface"
   // VAR_INPUT
   //    enable : Bool;
   //    selectTeachingPos : SInt;
   //    indexTeachingPos : SInt;
   // END_VAR
   // VAR_IN_OUT
   //    configurationSetPositions : Array[0..15] of "LBC_typeAxis64PosSetPosition";
   //    moduleInterface : "LBC_typeAxis64PosInterface";
   //    hmiInterface : Array[0..48] of "LER_TypeTeachingPosInterface";
   // END_VAR
   // VAR
   //    statPulse : Array[0..9] of Bool;
   //    statTonTimer : Array[0..15] of TON_TIME;
   //    statLastTeachingPosIndex : SInt;
   // END_VAR
BEGIN
END_DATA_BLOCK

DATA_BLOCK "instTeachingPosCathodeAlignTableAxisY2"   // DB464
// stored: InstanceOfName LER_TeachingPos_Interface, InstanceOfType FB
"LER_TeachingPos_Interface"
   // VAR_INPUT
   //    enable : Bool;
   //    selectTeachingPos : SInt;
   //    indexTeachingPos : SInt;
   // END_VAR
   // VAR_IN_OUT
   //    configurationSetPositions : Array[0..15] of "LBC_typeAxis64PosSetPosition";
   //    moduleInterface : "LBC_typeAxis64PosInterface";
   //    hmiInterface : Array[0..48] of "LER_TypeTeachingPosInterface";
   // END_VAR
   // VAR
   //    statPulse : Array[0..9] of Bool;
   //    statTonTimer : Array[0..15] of TON_TIME;
   //    statLastTeachingPosIndex : SInt;
   // END_VAR
BEGIN
END_DATA_BLOCK

DATA_BLOCK "instTeachingPosCathodeMainPnP1AxisX"   // DB278
// stored: InstanceOfName LER_TeachingPos_Interface, InstanceOfType FB
"LER_TeachingPos_Interface"
   // VAR_INPUT
   //    enable : Bool;
   //    selectTeachingPos : SInt;
   //    indexTeachingPos : SInt;
   // END_VAR
   // VAR_IN_OUT
   //    configurationSetPositions : Array[0..15] of "LBC_typeAxis64PosSetPosition";
   //    moduleInterface : "LBC_typeAxis64PosInterface";
   //    hmiInterface : Array[0..48] of "LER_TypeTeachingPosInterface";
   // END_VAR
   // VAR
   //    statPulse : Array[0..9] of Bool;
   //    statTonTimer : Array[0..15] of TON_TIME;
   //    statLastTeachingPosIndex : SInt;
   // END_VAR
BEGIN
END_DATA_BLOCK

DATA_BLOCK "instTeachingPosCathodeMainPnP1AxisY"   // DB353
// stored: InstanceOfName LER_TeachingPos_Interface, InstanceOfType FB
"LER_TeachingPos_Interface"
   // VAR_INPUT
   //    enable : Bool;
   //    selectTeachingPos : SInt;
   //    indexTeachingPos : SInt;
   // END_VAR
   // VAR_IN_OUT
   //    configurationSetPositions : Array[0..15] of "LBC_typeAxis64PosSetPosition";
   //    moduleInterface : "LBC_typeAxis64PosInterface";
   //    hmiInterface : Array[0..48] of "LER_TypeTeachingPosInterface";
   // END_VAR
   // VAR
   //    statPulse : Array[0..9] of Bool;
   //    statTonTimer : Array[0..15] of TON_TIME;
   //    statLastTeachingPosIndex : SInt;
   // END_VAR
BEGIN
END_DATA_BLOCK

DATA_BLOCK "instTeachingPosCathodeMainPnP1AxisZ"   // DB354
// stored: InstanceOfName LER_TeachingPos_Interface, InstanceOfType FB
"LER_TeachingPos_Interface"
   // VAR_INPUT
   //    enable : Bool;
   //    selectTeachingPos : SInt;
   //    indexTeachingPos : SInt;
   // END_VAR
   // VAR_IN_OUT
   //    configurationSetPositions : Array[0..15] of "LBC_typeAxis64PosSetPosition";
   //    moduleInterface : "LBC_typeAxis64PosInterface";
   //    hmiInterface : Array[0..48] of "LER_TypeTeachingPosInterface";
   // END_VAR
   // VAR
   //    statPulse : Array[0..9] of Bool;
   //    statTonTimer : Array[0..15] of TON_TIME;
   //    statLastTeachingPosIndex : SInt;
   // END_VAR
BEGIN
END_DATA_BLOCK

DATA_BLOCK "instTeachingPosCathodeMainPnP2AxisX"   // DB352
// stored: InstanceOfName LER_TeachingPos_Interface, InstanceOfType FB
"LER_TeachingPos_Interface"
   // VAR_INPUT
   //    enable : Bool;
   //    selectTeachingPos : SInt;
   //    indexTeachingPos : SInt;
   // END_VAR
   // VAR_IN_OUT
   //    configurationSetPositions : Array[0..15] of "LBC_typeAxis64PosSetPosition";
   //    moduleInterface : "LBC_typeAxis64PosInterface";
   //    hmiInterface : Array[0..48] of "LER_TypeTeachingPosInterface";
   // END_VAR
   // VAR
   //    statPulse : Array[0..9] of Bool;
   //    statTonTimer : Array[0..15] of TON_TIME;
   //    statLastTeachingPosIndex : SInt;
   // END_VAR
BEGIN
END_DATA_BLOCK

DATA_BLOCK "instTeachingPosCathodeMainPnP2AxisZ"   // DB451
// stored: InstanceOfName LER_TeachingPos_Interface, InstanceOfType FB
"LER_TeachingPos_Interface"
   // VAR_INPUT
   //    enable : Bool;
   //    selectTeachingPos : SInt;
   //    indexTeachingPos : SInt;
   // END_VAR
   // VAR_IN_OUT
   //    configurationSetPositions : Array[0..15] of "LBC_typeAxis64PosSetPosition";
   //    moduleInterface : "LBC_typeAxis64PosInterface";
   //    hmiInterface : Array[0..48] of "LER_TypeTeachingPosInterface";
   // END_VAR
   // VAR
   //    statPulse : Array[0..9] of Bool;
   //    statTonTimer : Array[0..15] of TON_TIME;
   //    statLastTeachingPosIndex : SInt;
   // END_VAR
BEGIN
END_DATA_BLOCK

DATA_BLOCK "instTeachingPosCompensatorAxisX"   // DB270
// stored: InstanceOfName LER_TeachingPos_Interface, InstanceOfType FB
"LER_TeachingPos_Interface"
   // VAR_INPUT
   //    enable : Bool;
   //    selectTeachingPos : SInt;
   //    indexTeachingPos : SInt;
   // END_VAR
   // VAR_IN_OUT
   //    configurationSetPositions : Array[0..15] of "LBC_typeAxis64PosSetPosition";
   //    moduleInterface : "LBC_typeAxis64PosInterface";
   //    hmiInterface : Array[0..48] of "LER_TypeTeachingPosInterface";
   // END_VAR
   // VAR
   //    statPulse : Array[0..9] of Bool;
   //    statTonTimer : Array[0..15] of TON_TIME;
   //    statLastTeachingPosIndex : SInt;
   // END_VAR
BEGIN
END_DATA_BLOCK

DATA_BLOCK "instTeachingPosFinalRollerFrontAxisX"   // DB465
// stored: InstanceOfName LER_TeachingPos_Interface, InstanceOfType FB
"LER_TeachingPos_Interface"
   // VAR_INPUT
   //    enable : Bool;
   //    selectTeachingPos : SInt;
   //    indexTeachingPos : SInt;
   // END_VAR
   // VAR_IN_OUT
   //    configurationSetPositions : Array[0..15] of "LBC_typeAxis64PosSetPosition";
   //    moduleInterface : "LBC_typeAxis64PosInterface";
   //    hmiInterface : Array[0..48] of "LER_TypeTeachingPosInterface";
   // END_VAR
   // VAR
   //    statPulse : Array[0..9] of Bool;
   //    statTonTimer : Array[0..15] of TON_TIME;
   //    statLastTeachingPosIndex : SInt;
   // END_VAR
BEGIN
END_DATA_BLOCK

DATA_BLOCK "instTeachingPosFinalRollerRearAxisX"   // DB466
// stored: InstanceOfName LER_TeachingPos_Interface, InstanceOfType FB
"LER_TeachingPos_Interface"
   // VAR_INPUT
   //    enable : Bool;
   //    selectTeachingPos : SInt;
   //    indexTeachingPos : SInt;
   // END_VAR
   // VAR_IN_OUT
   //    configurationSetPositions : Array[0..15] of "LBC_typeAxis64PosSetPosition";
   //    moduleInterface : "LBC_typeAxis64PosInterface";
   //    hmiInterface : Array[0..48] of "LER_TypeTeachingPosInterface";
   // END_VAR
   // VAR
   //    statPulse : Array[0..9] of Bool;
   //    statTonTimer : Array[0..15] of TON_TIME;
   //    statLastTeachingPosIndex : SInt;
   // END_VAR
BEGIN
END_DATA_BLOCK

DATA_BLOCK "instTeachingPosJRWinderAxisB"   // DB485
// stored: InstanceOfName LER_TeachingPos_Interface, InstanceOfType FB
"LER_TeachingPos_Interface"
   // VAR_INPUT
   //    enable : Bool;
   //    selectTeachingPos : SInt;
   //    indexTeachingPos : SInt;
   // END_VAR
   // VAR_IN_OUT
   //    configurationSetPositions : Array[0..15] of "LBC_typeAxis64PosSetPosition";
   //    moduleInterface : "LBC_typeAxis64PosInterface";
   //    hmiInterface : Array[0..48] of "LER_TypeTeachingPosInterface";
   // END_VAR
   // VAR
   //    statPulse : Array[0..9] of Bool;
   //    statTonTimer : Array[0..15] of TON_TIME;
   //    statLastTeachingPosIndex : SInt;
   // END_VAR
BEGIN
END_DATA_BLOCK

DATA_BLOCK "instTeachingPosJRWinderFrontAxisY"   // DB484
// stored: InstanceOfName LER_TeachingPos_Interface, InstanceOfType FB
"LER_TeachingPos_Interface"
   // VAR_INPUT
   //    enable : Bool;
   //    selectTeachingPos : SInt;
   //    indexTeachingPos : SInt;
   // END_VAR
   // VAR_IN_OUT
   //    configurationSetPositions : Array[0..15] of "LBC_typeAxis64PosSetPosition";
   //    moduleInterface : "LBC_typeAxis64PosInterface";
   //    hmiInterface : Array[0..48] of "LER_TypeTeachingPosInterface";
   // END_VAR
   // VAR
   //    statPulse : Array[0..9] of Bool;
   //    statTonTimer : Array[0..15] of TON_TIME;
   //    statLastTeachingPosIndex : SInt;
   // END_VAR
BEGIN
END_DATA_BLOCK

DATA_BLOCK "instTeachingPosJRWinderRearAxisY"   // DB483
// stored: InstanceOfName LER_TeachingPos_Interface, InstanceOfType FB
"LER_TeachingPos_Interface"
   // VAR_INPUT
   //    enable : Bool;
   //    selectTeachingPos : SInt;
   //    indexTeachingPos : SInt;
   // END_VAR
   // VAR_IN_OUT
   //    configurationSetPositions : Array[0..15] of "LBC_typeAxis64PosSetPosition";
   //    moduleInterface : "LBC_typeAxis64PosInterface";
   //    hmiInterface : Array[0..48] of "LER_TypeTeachingPosInterface";
   // END_VAR
   // VAR
   //    statPulse : Array[0..9] of Bool;
   //    statTonTimer : Array[0..15] of TON_TIME;
   //    statLastTeachingPosIndex : SInt;
   // END_VAR
BEGIN
END_DATA_BLOCK

DATA_BLOCK "instTeachingPosMendrelAnodeFrontAxisY"   // DB467
// stored: InstanceOfName LER_TeachingPos_Interface, InstanceOfType FB
"LER_TeachingPos_Interface"
   // VAR_INPUT
   //    enable : Bool;
   //    selectTeachingPos : SInt;
   //    indexTeachingPos : SInt;
   // END_VAR
   // VAR_IN_OUT
   //    configurationSetPositions : Array[0..15] of "LBC_typeAxis64PosSetPosition";
   //    moduleInterface : "LBC_typeAxis64PosInterface";
   //    hmiInterface : Array[0..48] of "LER_TypeTeachingPosInterface";
   // END_VAR
   // VAR
   //    statPulse : Array[0..9] of Bool;
   //    statTonTimer : Array[0..15] of TON_TIME;
   //    statLastTeachingPosIndex : SInt;
   // END_VAR
BEGIN
END_DATA_BLOCK

DATA_BLOCK "instTeachingPosMendrelAnodeFrontAxisZ"   // DB468
// stored: InstanceOfName LER_TeachingPos_Interface, InstanceOfType FB
"LER_TeachingPos_Interface"
   // VAR_INPUT
   //    enable : Bool;
   //    selectTeachingPos : SInt;
   //    indexTeachingPos : SInt;
   // END_VAR
   // VAR_IN_OUT
   //    configurationSetPositions : Array[0..15] of "LBC_typeAxis64PosSetPosition";
   //    moduleInterface : "LBC_typeAxis64PosInterface";
   //    hmiInterface : Array[0..48] of "LER_TypeTeachingPosInterface";
   // END_VAR
   // VAR
   //    statPulse : Array[0..9] of Bool;
   //    statTonTimer : Array[0..15] of TON_TIME;
   //    statLastTeachingPosIndex : SInt;
   // END_VAR
BEGIN
END_DATA_BLOCK

DATA_BLOCK "instTeachingPosMendrelAnodeRearAxisY"   // DB469
// stored: InstanceOfName LER_TeachingPos_Interface, InstanceOfType FB
"LER_TeachingPos_Interface"
   // VAR_INPUT
   //    enable : Bool;
   //    selectTeachingPos : SInt;
   //    indexTeachingPos : SInt;
   // END_VAR
   // VAR_IN_OUT
   //    configurationSetPositions : Array[0..15] of "LBC_typeAxis64PosSetPosition";
   //    moduleInterface : "LBC_typeAxis64PosInterface";
   //    hmiInterface : Array[0..48] of "LER_TypeTeachingPosInterface";
   // END_VAR
   // VAR
   //    statPulse : Array[0..9] of Bool;
   //    statTonTimer : Array[0..15] of TON_TIME;
   //    statLastTeachingPosIndex : SInt;
   // END_VAR
BEGIN
END_DATA_BLOCK

DATA_BLOCK "instTeachingPosMendrelAnodeRearAxisZ"   // DB470
// stored: InstanceOfName LER_TeachingPos_Interface, InstanceOfType FB
"LER_TeachingPos_Interface"
   // VAR_INPUT
   //    enable : Bool;
   //    selectTeachingPos : SInt;
   //    indexTeachingPos : SInt;
   // END_VAR
   // VAR_IN_OUT
   //    configurationSetPositions : Array[0..15] of "LBC_typeAxis64PosSetPosition";
   //    moduleInterface : "LBC_typeAxis64PosInterface";
   //    hmiInterface : Array[0..48] of "LER_TypeTeachingPosInterface";
   // END_VAR
   // VAR
   //    statPulse : Array[0..9] of Bool;
   //    statTonTimer : Array[0..15] of TON_TIME;
   //    statLastTeachingPosIndex : SInt;
   // END_VAR
BEGIN
END_DATA_BLOCK

DATA_BLOCK "instTeachingPosMendrelCathodeFrontAxisY"   // DB471
// stored: InstanceOfName LER_TeachingPos_Interface, InstanceOfType FB
"LER_TeachingPos_Interface"
   // VAR_INPUT
   //    enable : Bool;
   //    selectTeachingPos : SInt;
   //    indexTeachingPos : SInt;
   // END_VAR
   // VAR_IN_OUT
   //    configurationSetPositions : Array[0..15] of "LBC_typeAxis64PosSetPosition";
   //    moduleInterface : "LBC_typeAxis64PosInterface";
   //    hmiInterface : Array[0..48] of "LER_TypeTeachingPosInterface";
   // END_VAR
   // VAR
   //    statPulse : Array[0..9] of Bool;
   //    statTonTimer : Array[0..15] of TON_TIME;
   //    statLastTeachingPosIndex : SInt;
   // END_VAR
BEGIN
END_DATA_BLOCK

DATA_BLOCK "instTeachingPosMendrelCathodeFrontAxisZ"   // DB472
// stored: InstanceOfName LER_TeachingPos_Interface, InstanceOfType FB
"LER_TeachingPos_Interface"
   // VAR_INPUT
   //    enable : Bool;
   //    selectTeachingPos : SInt;
   //    indexTeachingPos : SInt;
   // END_VAR
   // VAR_IN_OUT
   //    configurationSetPositions : Array[0..15] of "LBC_typeAxis64PosSetPosition";
   //    moduleInterface : "LBC_typeAxis64PosInterface";
   //    hmiInterface : Array[0..48] of "LER_TypeTeachingPosInterface";
   // END_VAR
   // VAR
   //    statPulse : Array[0..9] of Bool;
   //    statTonTimer : Array[0..15] of TON_TIME;
   //    statLastTeachingPosIndex : SInt;
   // END_VAR
BEGIN
END_DATA_BLOCK

DATA_BLOCK "instTeachingPosMendrelCathodeRearAxisY"   // DB473
// stored: InstanceOfName LER_TeachingPos_Interface, InstanceOfType FB
"LER_TeachingPos_Interface"
   // VAR_INPUT
   //    enable : Bool;
   //    selectTeachingPos : SInt;
   //    indexTeachingPos : SInt;
   // END_VAR
   // VAR_IN_OUT
   //    configurationSetPositions : Array[0..15] of "LBC_typeAxis64PosSetPosition";
   //    moduleInterface : "LBC_typeAxis64PosInterface";
   //    hmiInterface : Array[0..48] of "LER_TypeTeachingPosInterface";
   // END_VAR
   // VAR
   //    statPulse : Array[0..9] of Bool;
   //    statTonTimer : Array[0..15] of TON_TIME;
   //    statLastTeachingPosIndex : SInt;
   // END_VAR
BEGIN
END_DATA_BLOCK

DATA_BLOCK "instTeachingPosMendrelCathodeRearAxisZ"   // DB474
// stored: InstanceOfName LER_TeachingPos_Interface, InstanceOfType FB
"LER_TeachingPos_Interface"
   // VAR_INPUT
   //    enable : Bool;
   //    selectTeachingPos : SInt;
   //    indexTeachingPos : SInt;
   // END_VAR
   // VAR_IN_OUT
   //    configurationSetPositions : Array[0..15] of "LBC_typeAxis64PosSetPosition";
   //    moduleInterface : "LBC_typeAxis64PosInterface";
   //    hmiInterface : Array[0..48] of "LER_TypeTeachingPosInterface";
   // END_VAR
   // VAR
   //    statPulse : Array[0..9] of Bool;
   //    statTonTimer : Array[0..15] of TON_TIME;
   //    statLastTeachingPosIndex : SInt;
   // END_VAR
BEGIN
END_DATA_BLOCK

DATA_BLOCK "instTeachingPosSepaClampnCutterAxisX"   // DB478
// stored: InstanceOfName LER_TeachingPos_Interface, InstanceOfType FB
"LER_TeachingPos_Interface"
   // VAR_INPUT
   //    enable : Bool;
   //    selectTeachingPos : SInt;
   //    indexTeachingPos : SInt;
   // END_VAR
   // VAR_IN_OUT
   //    configurationSetPositions : Array[0..15] of "LBC_typeAxis64PosSetPosition";
   //    moduleInterface : "LBC_typeAxis64PosInterface";
   //    hmiInterface : Array[0..48] of "LER_TypeTeachingPosInterface";
   // END_VAR
   // VAR
   //    statPulse : Array[0..9] of Bool;
   //    statTonTimer : Array[0..15] of TON_TIME;
   //    statLastTeachingPosIndex : SInt;
   // END_VAR
BEGIN
END_DATA_BLOCK

DATA_BLOCK "instTeachingPosSepaClampnCutterAxisZ"   // DB479
// stored: InstanceOfName LER_TeachingPos_Interface, InstanceOfType FB
"LER_TeachingPos_Interface"
   // VAR_INPUT
   //    enable : Bool;
   //    selectTeachingPos : SInt;
   //    indexTeachingPos : SInt;
   // END_VAR
   // VAR_IN_OUT
   //    configurationSetPositions : Array[0..15] of "LBC_typeAxis64PosSetPosition";
   //    moduleInterface : "LBC_typeAxis64PosInterface";
   //    hmiInterface : Array[0..48] of "LER_TypeTeachingPosInterface";
   // END_VAR
   // VAR
   //    statPulse : Array[0..9] of Bool;
   //    statTonTimer : Array[0..15] of TON_TIME;
   //    statLastTeachingPosIndex : SInt;
   // END_VAR
BEGIN
END_DATA_BLOCK

DATA_BLOCK "instTeachingPosSepaGripperAxisC"   // DB482
// stored: InstanceOfName LER_TeachingPos_Interface, InstanceOfType FB
"LER_TeachingPos_Interface"
   // VAR_INPUT
   //    enable : Bool;
   //    selectTeachingPos : SInt;
   //    indexTeachingPos : SInt;
   // END_VAR
   // VAR_IN_OUT
   //    configurationSetPositions : Array[0..15] of "LBC_typeAxis64PosSetPosition";
   //    moduleInterface : "LBC_typeAxis64PosInterface";
   //    hmiInterface : Array[0..48] of "LER_TypeTeachingPosInterface";
   // END_VAR
   // VAR
   //    statPulse : Array[0..9] of Bool;
   //    statTonTimer : Array[0..15] of TON_TIME;
   //    statLastTeachingPosIndex : SInt;
   // END_VAR
BEGIN
END_DATA_BLOCK

DATA_BLOCK "instTeachingPosSepaGripperAxisX"   // DB480
// stored: InstanceOfName LER_TeachingPos_Interface, InstanceOfType FB
"LER_TeachingPos_Interface"
   // VAR_INPUT
   //    enable : Bool;
   //    selectTeachingPos : SInt;
   //    indexTeachingPos : SInt;
   // END_VAR
   // VAR_IN_OUT
   //    configurationSetPositions : Array[0..15] of "LBC_typeAxis64PosSetPosition";
   //    moduleInterface : "LBC_typeAxis64PosInterface";
   //    hmiInterface : Array[0..48] of "LER_TypeTeachingPosInterface";
   // END_VAR
   // VAR
   //    statPulse : Array[0..9] of Bool;
   //    statTonTimer : Array[0..15] of TON_TIME;
   //    statLastTeachingPosIndex : SInt;
   // END_VAR
BEGIN
END_DATA_BLOCK

DATA_BLOCK "instTeachingPosSepaGripperAxisZ"   // DB481
// stored: InstanceOfName LER_TeachingPos_Interface, InstanceOfType FB
"LER_TeachingPos_Interface"
   // VAR_INPUT
   //    enable : Bool;
   //    selectTeachingPos : SInt;
   //    indexTeachingPos : SInt;
   // END_VAR
   // VAR_IN_OUT
   //    configurationSetPositions : Array[0..15] of "LBC_typeAxis64PosSetPosition";
   //    moduleInterface : "LBC_typeAxis64PosInterface";
   //    hmiInterface : Array[0..48] of "LER_TypeTeachingPosInterface";
   // END_VAR
   // VAR
   //    statPulse : Array[0..9] of Bool;
   //    statTonTimer : Array[0..15] of TON_TIME;
   //    statLastTeachingPosIndex : SInt;
   // END_VAR
BEGIN
END_DATA_BLOCK

DATA_BLOCK "instTeachingPosStackTableOutFrontAxisZ"   // DB476
// stored: InstanceOfName LER_TeachingPos_Interface, InstanceOfType FB
"LER_TeachingPos_Interface"
   // VAR_INPUT
   //    enable : Bool;
   //    selectTeachingPos : SInt;
   //    indexTeachingPos : SInt;
   // END_VAR
   // VAR_IN_OUT
   //    configurationSetPositions : Array[0..15] of "LBC_typeAxis64PosSetPosition";
   //    moduleInterface : "LBC_typeAxis64PosInterface";
   //    hmiInterface : Array[0..48] of "LER_TypeTeachingPosInterface";
   // END_VAR
   // VAR
   //    statPulse : Array[0..9] of Bool;
   //    statTonTimer : Array[0..15] of TON_TIME;
   //    statLastTeachingPosIndex : SInt;
   // END_VAR
BEGIN
END_DATA_BLOCK

DATA_BLOCK "instTeachingPosStackTableOutRearAxisZ"   // DB477
// stored: InstanceOfName LER_TeachingPos_Interface, InstanceOfType FB
"LER_TeachingPos_Interface"
   // VAR_INPUT
   //    enable : Bool;
   //    selectTeachingPos : SInt;
   //    indexTeachingPos : SInt;
   // END_VAR
   // VAR_IN_OUT
   //    configurationSetPositions : Array[0..15] of "LBC_typeAxis64PosSetPosition";
   //    moduleInterface : "LBC_typeAxis64PosInterface";
   //    hmiInterface : Array[0..48] of "LER_TypeTeachingPosInterface";
   // END_VAR
   // VAR
   //    statPulse : Array[0..9] of Bool;
   //    statTonTimer : Array[0..15] of TON_TIME;
   //    statLastTeachingPosIndex : SInt;
   // END_VAR
BEGIN
END_DATA_BLOCK

DATA_BLOCK "instTeachingPosStackTableZ"   // DB475
// stored: InstanceOfName LER_TeachingPos_Interface, InstanceOfType FB
"LER_TeachingPos_Interface"
   // VAR_INPUT
   //    enable : Bool;
   //    selectTeachingPos : SInt;
   //    indexTeachingPos : SInt;
   // END_VAR
   // VAR_IN_OUT
   //    configurationSetPositions : Array[0..15] of "LBC_typeAxis64PosSetPosition";
   //    moduleInterface : "LBC_typeAxis64PosInterface";
   //    hmiInterface : Array[0..48] of "LER_TypeTeachingPosInterface";
   // END_VAR
   // VAR
   //    statPulse : Array[0..9] of Bool;
   //    statTonTimer : Array[0..15] of TON_TIME;
   //    statLastTeachingPosIndex : SInt;
   // END_VAR
BEGIN
END_DATA_BLOCK

DATA_BLOCK "instTeachingPosUnwinderBottomAxisB"   // DB269
// stored: InstanceOfName LER_TeachingPos_Interface, InstanceOfType FB
"LER_TeachingPos_Interface"
   // VAR_INPUT
   //    enable : Bool;
   //    selectTeachingPos : SInt;
   //    indexTeachingPos : SInt;
   // END_VAR
   // VAR_IN_OUT
   //    configurationSetPositions : Array[0..15] of "LBC_typeAxis64PosSetPosition";
   //    moduleInterface : "LBC_typeAxis64PosInterface";
   //    hmiInterface : Array[0..48] of "LER_TypeTeachingPosInterface";
   // END_VAR
   // VAR
   //    statPulse : Array[0..9] of Bool;
   //    statTonTimer : Array[0..15] of TON_TIME;
   //    statLastTeachingPosIndex : SInt;
   // END_VAR
BEGIN
END_DATA_BLOCK

DATA_BLOCK "instTeachingPosUnwinderTopAxisB"   // DB268
// stored: InstanceOfName LER_TeachingPos_Interface, InstanceOfType FB
"LER_TeachingPos_Interface"
   // VAR_INPUT
   //    enable : Bool;
   //    selectTeachingPos : SInt;
   //    indexTeachingPos : SInt;
   // END_VAR
   // VAR_IN_OUT
   //    configurationSetPositions : Array[0..15] of "LBC_typeAxis64PosSetPosition";
   //    moduleInterface : "LBC_typeAxis64PosInterface";
   //    hmiInterface : Array[0..48] of "LER_TypeTeachingPosInterface";
   // END_VAR
   // VAR
   //    statPulse : Array[0..9] of Bool;
   //    statTonTimer : Array[0..15] of TON_TIME;
   //    statLastTeachingPosIndex : SInt;
   // END_VAR
BEGIN
END_DATA_BLOCK

DATA_BLOCK "InstGetAxisStatus"   // DB2
AUTHOR : Siemens Digital Industries
FAMILY : LAF
NAME : LAF_GetAxisStatus
VERSION : 1.1
// stored: InstanceOfName LAF_GetAxisStatus, InstanceOfType FB
"LAF_GetAxisStatus"
   // VAR_INPUT
   //    enable : Bool := TRUE;
   // END_VAR
   // VAR_OUTPUT
   //    valid { ExternalWritable := 'False'} : Bool := FALSE;
   //    busy { ExternalWritable := 'False'} : Bool := FALSE;
   //    error { ExternalWritable := 'False'} : Bool := FALSE;
   //    status { ExternalWritable := 'False'} : Word := 16#7000;
   //    diagnostics { ExternalWritable := 'False'} : "LAF_typeDiagnostics";
   // END_VAR
   // VAR_IN_OUT
   //    configuration : Array[*] of "LAF_typeDriveDiagConfig";
   //    moduleInterface : "LAF_typeDriveDiagInterfaceHmi";
   // END_VAR
   // VAR
   //    statInternal { ExternalAccessible := 'False'; ExternalVisible := 'False'; ExternalWritable := 'False'} : Struct
   //       enablePrevious : Bool := FALSE;
   //       valid : Bool := FALSE;
   //       busy : Bool := FALSE;
   //       error : Bool := FALSE;
   //       errorUserCleared : Bool := FALSE;
   //       errorAutoCleared : Bool := FALSE;
   //       disablingCompleted : Bool := TRUE;
   //       diagnostics : "LAF_typeDiagnostics";
   //       emptyDiagnostics : "LAF_typeDiagnostics";
   //    END_STRUCT;
   //    statMainState { ExternalAccessible := 'False'; ExternalVisible := 'False'; ExternalWritable := 'False'} : DInt := 0;
   //    statArrayMin { ExternalAccessible := 'False'; ExternalVisible := 'False'; ExternalWritable := 'False'} : DInt := 0;
   //    statArrayMax { ExternalAccessible := 'False'; ExternalVisible := 'False'; ExternalWritable := 'False'} : DInt := 41;
   // END_VAR
BEGIN
   diagnostics.status := 16#7000;
   diagnostics.subfunctionStatus := 16#0000;
   diagnostics.stateNumber := 0;
   statInternal.diagnostics.status := 16#7000;
   statInternal.diagnostics.subfunctionStatus := 16#0000;
   statInternal.diagnostics.stateNumber := 50;
   statInternal.emptyDiagnostics.status := 16#7000;
   statInternal.emptyDiagnostics.subfunctionStatus := 16#0000;
   statInternal.emptyDiagnostics.stateNumber := 0;
END_DATA_BLOCK

DATA_BLOCK "InstGetSinaAlarms"   // DB74
AUTHOR : Siemens Digital Industries
FAMILY : LAF
NAME : LAF_GetSinaAlarms
VERSION : 1.1
// stored: InstanceOfName LAF_GetSinaAlarms, InstanceOfType FB
"LAF_GetSinaAlarms"
   // VAR_INPUT
   //    enable : Bool := TRUE;
   // END_VAR
   // VAR_OUTPUT
   //    valid { ExternalWritable := 'False'} : Bool := FALSE;
   //    busy { ExternalWritable := 'False'} : Bool := FALSE;
   //    error { ExternalWritable := 'False'} : Bool := FALSE;
   //    status { ExternalWritable := 'False'} : Word := 16#7000;
   //    diagnostics { ExternalWritable := 'False'} : "LAF_typeDiagnostics";
   //    statusWriteRecord { ExternalWritable := 'False'} : DWord := 16#0000_0000;
   //    statusReadRecord { ExternalWritable := 'False'} : DWord := 16#0000_0000;
   // END_VAR
   // VAR_IN_OUT
   //    configuration : Array[*] of "LAF_typeDriveDiagConfig";
   //    moduleInterface : "LAF_typeDriveDiagInterfaceHmi";
   // END_VAR
   // VAR
   //    statInternal { ExternalAccessible := 'False'; ExternalVisible := 'False'; ExternalWritable := 'False'} : Struct
   //       enablePrevious : Bool := FALSE;
   //       valid : Bool := FALSE;
   //       busy : Bool := FALSE;
   //       error : Bool := FALSE;
   //       errorUserCleared : Bool := FALSE;
   //       errorAutoCleared : Bool := FALSE;
   //       disablingCompleted : Bool := FALSE;
   //       diagnostics : "LAF_typeDiagnostics";
   //       emptyDiagnostics : "LAF_typeDiagnostics";
   //    END_STRUCT;
   //    statMainState { ExternalAccessible := 'False'; ExternalVisible := 'False'; ExternalWritable := 'False'} : DInt := 0;
   //    statArrayMin { ExternalAccessible := 'False'; ExternalVisible := 'False'; ExternalWritable := 'False'} : DInt := 0;
   //    statArrayMax { ExternalAccessible := 'False'; ExternalVisible := 'False'; ExternalWritable := 'False'} : DInt := 0;
   //    instWriteRecord { ExternalAccessible := 'False'; ExternalVisible := 'False'; ExternalWritable := 'False'} : WRREC;
   //    instReadRecord { ExternalAccessible := 'False'; ExternalVisible := 'False'; ExternalWritable := 'False'} : RDREC;
   //    statWriteReq { ExternalAccessible := 'False'; ExternalVisible := 'False'; ExternalWritable := 'False'} : Struct
   //       header : Struct
   //          reqRef : Byte := 16#00;
   //          reqID : Byte := 16#00;
   //          axis : Byte := 16#01;
   //          noPara : Byte := 16#01;
   //       END_STRUCT;
   //       data : Array[0..235] of Byte;
   //    END_STRUCT;
   //    statReadReq { ExternalAccessible := 'False'; ExternalVisible := 'False'; ExternalWritable := 'False'} : Struct
   //       header : Struct
   //          reqRef : Byte := 16#00;
   //          reqID : Byte := 16#00;
   //          axis : Byte := 16#01;
   //          noPara : Byte := 16#01;
   //       END_STRUCT;
   //       data : Array[0..235] of Byte;
   //    END_STRUCT;
   //    instActTimer { ExternalAccessible := 'False'; ExternalVisible := 'False'; ExternalWritable := 'False'} : IEC_TIMER;
   //    instReqTimer { ExternalAccessible := 'False'; ExternalVisible := 'False'; ExternalWritable := 'False'} : IEC_TIMER;
   //    statDataTransRun { ExternalAccessible := 'False'; ExternalVisible := 'False'; ExternalWritable := 'False'} : Bool := FALSE;
   //    statWriteReqSet { ExternalAccessible := 'False'; ExternalVisible := 'False'; ExternalWritable := 'False'} : Bool := FALSE;
   //    statActTimerIn { ExternalAccessible := 'False'; ExternalVisible := 'False'; ExternalWritable := 'False'} : Bool := FALSE;
   //    statPrevTimeValue { ExternalAccessible := 'False'; ExternalVisible := 'False'; ExternalWritable := 'False'} : Time := T#0MS;
   //    statActTimerValueAct { ExternalAccessible := 'False'; ExternalVisible := 'False'; ExternalWritable := 'False'} : Time := T#0MS;
   //    statActTimerValueReq { ExternalAccessible := 'False'; ExternalVisible := 'False'; ExternalWritable := 'False'} : Time := T#0MS;
   //    statPrevDriveIndex { ExternalAccessible := 'False'; ExternalVisible := 'False'; ExternalWritable := 'False'} : DInt := 0;
   // END_VAR
BEGIN
   diagnostics.status := 16#0000;
   diagnostics.subfunctionStatus := 16#0000;
   diagnostics.stateNumber := 0;
   statInternal.diagnostics.status := 16#7000;
   statInternal.diagnostics.subfunctionStatus := 16#0000;
   statInternal.diagnostics.stateNumber := 0;
   statInternal.emptyDiagnostics.status := 16#7000;
   statInternal.emptyDiagnostics.subfunctionStatus := 16#0000;
   statInternal.emptyDiagnostics.stateNumber := 0;
   instWriteRecord.REQ := FALSE;
   instWriteRecord.ID := 0;
   instWriteRecord.INDEX := 0;
   instWriteRecord.LEN := 0;
   instWriteRecord.DONE := FALSE;
   instWriteRecord.BUSY := FALSE;
   instWriteRecord.ERROR := FALSE;
   instWriteRecord.STATUS := 16#0000_0000;
   instReadRecord.REQ := FALSE;
   instReadRecord.ID := 0;
   instReadRecord.INDEX := 0;
   instReadRecord.MLEN := 0;
   instReadRecord.VALID := FALSE;
   instReadRecord.BUSY := FALSE;
   instReadRecord.ERROR := FALSE;
   instReadRecord.STATUS := 16#0000_0000;
   instReadRecord.LEN := 0;
   statWriteReq.data[0..235] := 16#00;
   statReadReq.data[0..235] := 16#00;
   instActTimer.PT := T#0MS;
   instActTimer.IN := FALSE;
   instReqTimer.PT := T#0MS;
   instReqTimer.IN := FALSE;
END_DATA_BLOCK

DATA_BLOCK "InstGetSinaEpos"   // DB86
AUTHOR : Siemens Digital Industries
FAMILY : LAF
NAME : LAF_GetSinaEpos
VERSION : 1.1
// stored: InstanceOfName LAF_GetSinaEpos, InstanceOfType FB
"LAF_GetSinaEpos"
   // VAR_INPUT
   //    enable : Bool := TRUE;
   // END_VAR
   // VAR_OUTPUT
   //    valid { ExternalWritable := 'False'} : Bool := FALSE;
   //    busy { ExternalWritable := 'False'} : Bool := FALSE;
   //    error { ExternalWritable := 'False'} : Bool := FALSE;
   //    status { ExternalWritable := 'False'} : Word := 16#7000;
   //    diagnostics { ExternalWritable := 'False'} : "LAF_typeDiagnostics";
   //    statusWriteRecord { ExternalAccessible := 'False'; ExternalVisible := 'False'; ExternalWritable := 'False'} : DWord := 16#0000_0000;
   //    statusReadRecord { ExternalAccessible := 'False'; ExternalVisible := 'False'; ExternalWritable := 'False'} : DWord := 16#0000_0000;
   // END_VAR
   // VAR_IN_OUT
   //    configuration : Array[*] of "LAF_typeDriveDiagConfig";
   //    moduleInterface : "LAF_typeDriveDiagInterfaceHmi";
   // END_VAR
   // VAR
   //    statInternal { ExternalAccessible := 'False'; ExternalVisible := 'False'; ExternalWritable := 'False'} : Struct
   //       enablePrevious : Bool := FALSE;
   //       valid : Bool := FALSE;
   //       busy : Bool := FALSE;
   //       error : Bool := FALSE;
   //       errorUserCleared : Bool := FALSE;
   //       errorAutoCleared : Bool := FALSE;
   //       disablingCompleted : Bool := FALSE;
   //       diagnostics : "LAF_typeDiagnostics";
   //       emptyDiagnostics : "LAF_typeDiagnostics";
   //    END_STRUCT;
   //    statMainState { ExternalAccessible := 'False'; ExternalVisible := 'False'; ExternalWritable := 'False'} : DInt := 0;
   //    statArrayMin { ExternalAccessible := 'False'; ExternalVisible := 'False'; ExternalWritable := 'False'} : DInt := 0;
   //    statArrayMax { ExternalAccessible := 'False'; ExternalVisible := 'False'; ExternalWritable := 'False'} : DInt := 0;
   //    instWriteRecord { ExternalAccessible := 'False'; ExternalVisible := 'False'; ExternalWritable := 'False'} : WRREC;
   //    instReadRecord { ExternalAccessible := 'False'; ExternalVisible := 'False'; ExternalWritable := 'False'} : RDREC;
   //    statWriteReq { ExternalAccessible := 'False'; ExternalVisible := 'False'; ExternalWritable := 'False'} : Struct
   //       header : Struct
   //          reqRef : Byte := 16#00;
   //          reqID : Byte := 16#00;
   //          axis : Byte := 16#01;
   //          noPara : Byte := 16#01;
   //       END_STRUCT;
   //       data : Array[0..235] of Byte;
   //    END_STRUCT;
   //    statReadReq { ExternalAccessible := 'False'; ExternalVisible := 'False'; ExternalWritable := 'False'} : Struct
   //       header : Struct
   //          reqRef : Byte := 16#00;
   //          reqID : Byte := 16#00;
   //          axis : Byte := 16#01;
   //          noPara : Byte := 16#01;
   //       END_STRUCT;
   //       data : Array[0..235] of Byte;
   //    END_STRUCT;
   //    instActTimer { ExternalAccessible := 'False'; ExternalVisible := 'False'; ExternalWritable := 'False'} : IEC_TIMER;
   //    instReqTimer { ExternalAccessible := 'False'; ExternalVisible := 'False'; ExternalWritable := 'False'} : IEC_TIMER;
   //    statDataTransRun { ExternalAccessible := 'False'; ExternalVisible := 'False'; ExternalWritable := 'False'} : Bool := FALSE;
   //    statWriteReqSet { ExternalAccessible := 'False'; ExternalVisible := 'False'; ExternalWritable := 'False'} : Bool := FALSE;
   //    statActTimerIn { ExternalAccessible := 'False'; ExternalVisible := 'False'; ExternalWritable := 'False'} : Bool := FALSE;
   //    statPrevTimeValue { ExternalAccessible := 'False'; ExternalVisible := 'False'; ExternalWritable := 'False'} : Time := T#0MS;
   //    statActTimerValueAct { ExternalAccessible := 'False'; ExternalVisible := 'False'; ExternalWritable := 'False'} : Time := T#0MS;
   //    statActTimerValueReq { ExternalAccessible := 'False'; ExternalVisible := 'False'; ExternalWritable := 'False'} : Time := T#0MS;
   //    statPrevDriveIndex { ExternalAccessible := 'False'; ExternalVisible := 'False'; ExternalWritable := 'False'} : DInt := 0;
   // END_VAR
BEGIN
   diagnostics.status := 16#0000;
   diagnostics.subfunctionStatus := 16#0000;
   diagnostics.stateNumber := 0;
   statInternal.diagnostics.status := 16#7000;
   statInternal.diagnostics.subfunctionStatus := 16#0000;
   statInternal.diagnostics.stateNumber := 0;
   statInternal.emptyDiagnostics.status := 16#7000;
   statInternal.emptyDiagnostics.subfunctionStatus := 16#0000;
   statInternal.emptyDiagnostics.stateNumber := 0;
   instWriteRecord.REQ := FALSE;
   instWriteRecord.ID := 0;
   instWriteRecord.INDEX := 0;
   instWriteRecord.LEN := 0;
   instWriteRecord.DONE := FALSE;
   instWriteRecord.BUSY := FALSE;
   instWriteRecord.ERROR := FALSE;
   instWriteRecord.STATUS := 16#0000_0000;
   instReadRecord.REQ := FALSE;
   instReadRecord.ID := 0;
   instReadRecord.INDEX := 0;
   instReadRecord.MLEN := 0;
   instReadRecord.VALID := FALSE;
   instReadRecord.BUSY := FALSE;
   instReadRecord.ERROR := FALSE;
   instReadRecord.STATUS := 16#0000_0000;
   instReadRecord.LEN := 0;
   statWriteReq.data[0..235] := 16#00;
   statReadReq.data[0..235] := 16#00;
   instActTimer.PT := T#0MS;
   instActTimer.IN := FALSE;
   instReqTimer.PT := T#0MS;
   instReqTimer.IN := FALSE;
END_DATA_BLOCK

DATA_BLOCK "InstGetSinaStatus"   // DB15
AUTHOR : Siemens Digital Industries
FAMILY : LAF
NAME : LAF_GetSinaStatus
VERSION : 1.1
// stored: InstanceOfName LAF_GetSinaStatus, InstanceOfType FB
"LAF_GetSinaStatus"
   // VAR_INPUT
   //    enable : Bool := TRUE;
   // END_VAR
   // VAR_OUTPUT
   //    valid { ExternalWritable := 'False'} : Bool := FALSE;
   //    busy { ExternalWritable := 'False'} : Bool := FALSE;
   //    error { ExternalWritable := 'False'} : Bool := FALSE;
   //    status { ExternalWritable := 'False'} : Word := 16#7000;
   //    diagnostics { ExternalWritable := 'False'} : "LAF_typeDiagnostics";
   //    statusWriteRecord { ExternalVisible := 'False'; ExternalWritable := 'False'} : DWord := 16#0000_0000;
   //    statusReadRecord { ExternalWritable := 'False'} : DWord := 16#0000_0000;
   // END_VAR
   // VAR_IN_OUT
   //    configuration : Array[*] of "LAF_typeDriveDiagConfig";
   //    moduleInterface : "LAF_typeDriveDiagInterfaceHmi";
   // END_VAR
   // VAR
   //    statInternal { ExternalAccessible := 'False'; ExternalVisible := 'False'; ExternalWritable := 'False'} : Struct
   //       enablePrevious : Bool := FALSE;
   //       valid : Bool := FALSE;
   //       busy : Bool := FALSE;
   //       error : Bool := FALSE;
   //       errorUserCleared : Bool := FALSE;
   //       errorAutoCleared : Bool := FALSE;
   //       disablingCompleted : Bool := FALSE;
   //       diagnostics : "LAF_typeDiagnostics";
   //       emptyDiagnostics : "LAF_typeDiagnostics";
   //    END_STRUCT;
   //    statMainState { ExternalAccessible := 'False'; ExternalVisible := 'False'; ExternalWritable := 'False'} : DInt := 0;
   //    statArrayMin { ExternalAccessible := 'False'; ExternalVisible := 'False'; ExternalWritable := 'False'} : DInt := 0;
   //    statArrayMax { ExternalAccessible := 'False'; ExternalVisible := 'False'; ExternalWritable := 'False'} : DInt := 0;
   //    instWriteRecord { ExternalAccessible := 'False'; ExternalVisible := 'False'; ExternalWritable := 'False'} : WRREC;
   //    instReadRecord { ExternalAccessible := 'False'; ExternalVisible := 'False'; ExternalWritable := 'False'} : RDREC;
   //    statWriteReq { ExternalAccessible := 'False'; ExternalVisible := 'False'; ExternalWritable := 'False'} : Struct
   //       header : Struct
   //          reqRef : Byte := 16#00;
   //          reqID : Byte := 16#00;
   //          axis : Byte := 16#01;
   //          noPara : Byte := 16#01;
   //       END_STRUCT;
   //       data : Array[0..235] of Byte;
   //    END_STRUCT;
   //    statReadReq { ExternalAccessible := 'False'; ExternalVisible := 'False'; ExternalWritable := 'False'} : Struct
   //       header : Struct
   //          reqRef : Byte := 16#00;
   //          reqID : Byte := 16#00;
   //          axis : Byte := 16#01;
   //          noPara : Byte := 16#01;
   //       END_STRUCT;
   //       data : Array[0..235] of Byte;
   //    END_STRUCT;
   //    instActTimer { ExternalAccessible := 'False'; ExternalVisible := 'False'; ExternalWritable := 'False'} : IEC_TIMER;
   //    instReqTimer { ExternalAccessible := 'False'; ExternalVisible := 'False'; ExternalWritable := 'False'} : IEC_TIMER;
   //    statDataTransRun { ExternalAccessible := 'False'; ExternalVisible := 'False'; ExternalWritable := 'False'} : Bool := FALSE;
   //    statWriteReqSet { ExternalAccessible := 'False'; ExternalVisible := 'False'; ExternalWritable := 'False'} : Bool := FALSE;
   //    statActTimerIn { ExternalAccessible := 'False'; ExternalVisible := 'False'; ExternalWritable := 'False'} : Bool := FALSE;
   //    statPrevTimeValue { ExternalAccessible := 'False'; ExternalVisible := 'False'; ExternalWritable := 'False'} : Time := T#0MS;
   //    statActTimerValueAct { ExternalAccessible := 'False'; ExternalVisible := 'False'; ExternalWritable := 'False'} : Time := T#0MS;
   //    statActTimerValueReq { ExternalAccessible := 'False'; ExternalVisible := 'False'; ExternalWritable := 'False'} : Time := T#0MS;
   //    statPrevDriveIndex { ExternalAccessible := 'False'; ExternalVisible := 'False'; ExternalWritable := 'False'} : DInt := 0;
   // END_VAR
BEGIN
   diagnostics.status := 16#0000;
   diagnostics.subfunctionStatus := 16#0000;
   diagnostics.stateNumber := 0;
   statInternal.diagnostics.status := 16#7000;
   statInternal.diagnostics.subfunctionStatus := 16#0000;
   statInternal.diagnostics.stateNumber := 0;
   statInternal.emptyDiagnostics.status := 16#7000;
   statInternal.emptyDiagnostics.subfunctionStatus := 16#0000;
   statInternal.emptyDiagnostics.stateNumber := 0;
   instWriteRecord.REQ := FALSE;
   instWriteRecord.ID := 0;
   instWriteRecord.INDEX := 0;
   instWriteRecord.LEN := 0;
   instWriteRecord.DONE := FALSE;
   instWriteRecord.BUSY := FALSE;
   instWriteRecord.ERROR := FALSE;
   instWriteRecord.STATUS := 16#0000_0000;
   instReadRecord.REQ := FALSE;
   instReadRecord.ID := 0;
   instReadRecord.INDEX := 0;
   instReadRecord.MLEN := 0;
   instReadRecord.VALID := FALSE;
   instReadRecord.BUSY := FALSE;
   instReadRecord.ERROR := FALSE;
   instReadRecord.STATUS := 16#0000_0000;
   instReadRecord.LEN := 0;
   statWriteReq.data[0..235] := 16#00;
   statReadReq.data[0..235] := 16#00;
   instActTimer.PT := T#0MS;
   instActTimer.IN := FALSE;
   instReqTimer.PT := T#0MS;
   instReqTimer.IN := FALSE;
END_DATA_BLOCK

